DATA_BLOCK "PDI"   // DB129
{ S7_Optimized_Access := 'FALSE' }
VERSION : 0.0
// --------------------------------------------------------------------------------
// program:             PDI
// description :        automatically generated PDI
// name:                hp
// date        :        03.02.2021
// 
// revision:
// name:
// date:
//                     (c)CGS
// --------------------------------------------------------------------------------
   VAR
      CB_FLT_DC24V_K2 : Bool;   // HDI def M 72.0: fault circuit breakers DC 24V 1=OK
      CB_FLT_AC400V_K2 : Bool;   // HDI def M 72.1: fault circuit breakers AC 400V 1=OK
      SPARE_16_2 : Bool;   // HDI def M 72.4: spare digital input
      CB_FLT_AC230V : Bool;   // HDI def M 72.3: fault circuit breakers AC 230V 1=OK
      SPARE_16_4 : Bool;   // HDI def M 72.4: spare digital input
      SPARE_16_5 : Bool;   // HDI def M 72.5: spare digital input
      SPARE_16_6 : Bool;   // HDI def M 72.6: spare digital input
      SPARE_16_7 : Bool;   // HDI def M 72.7: spare digital input
      SPARE_17_0 : Bool;   // HDI def M 73.0: spare digital input
      UPS_24V_ALM : Bool;   // HDI def M 73.1: alarm dc-usv
      UPS_24V_NRM : Bool;   // HDI def M 73.2: main line ready buffered dc-usv
      EMO : Bool;   // HDI def M 73.3: Emergency off (1=ok)
      EMS : Bool;   // HDI def M 73.4: Emergency stop handling drives (1=ok)
      SPARE_17_5 : Bool;   // HDI def M 73.5: spare digital input
      SPARE_17_6 : Bool;   // HDI def M 73.6: spare digital input
      SPARE_17_7 : Bool;   // HDI def M 73.7: spare digital input
      P1_WRN : Bool;   // HDI def M 74.0: pump unit (P1) warning
      P1_FLT : Bool;   // HDI def M 74.1: pump unit (P1) error
      P1_IS_ON : Bool;   // HDI def M 74.2: pump unit (P1) running
      P1_WD : Bool;   // HDI def M 74.3: pump unit (P1) watchdog
      FIL_APS : Bool;   // HDI def M 74.4: pressure filter 1000 mbar
      MON_TMP_P2 : Bool;   // HDI def M 74.5: temperature monitoring P2
      MON_TMP_P1 : Bool;   // HDI def M 74.6: temperature monitoring P1
      SPARE_18_7 : Bool;   // HDI def M 74.7: spare digital input
      FCH_LFT_SDL_NUT : Bool;   // HDI def M 88.0: safety limit switch furnace chamber lift spindle nut
      LS_FCH_LFT_DN : Bool;   // HDI def M 88.1: limit switch furnace chamber lift down
      LS_FCH_HOOK_WORK : Bool;   // HDI def M 88.2: limit switch furnace chamber hook in working position
      LS_FCH_HOOK_HOME : Bool;   // HDI def M 88.3: limit switch furnace chamber hook in home position
      LS_TEC_FLG_DN : Bool;   // HDI def M 88.4: limit switch technolgy flange down
      TEC_FLG_SDL_NUT : Bool;   // HDI def M 88.5: safety limit switch technolgy flange lift spindle nut
      LS_V11_COV_OP : Bool;   // HDI def M 88.6: Cover V11 opened (isolation valve feeder)
      LS_V11_COV_CL : Bool;   // HDI def M 88.7: Cover V11 closed (isolation valve feeder)
      GCH_APS : Bool;   // HDI def M 89.0: pressure gate chamber 1000 mbar
      FCH_APS : Bool;   // HDI def M 89.1: pressure furnace chamber 1000 mbar
      FDR_APS : Bool;   // HDI def M 89.2: pressure feeder 1000 mbar
      FIL_2_APS : Bool;   // HDI def M 89.3: atmospheric pressure filter 2
      SPARE_33_4 : Bool;   // HDI def M 89.4: spare
      SPARE_33_5 : Bool;   // HDI def M 89.5: spare
      LS_V2_1_OP : Bool;   // HDI def M 89.6: valve position v2.1 fce chamber
      LS_V2_1_CL : Bool;   // HDI def M 89.7: valve position v2.1 fce chamber
      CB_FLT_AC400V_K5 : Bool;   // HDI def M 90.0: fault circuit breakers AC 400V +K5 1=OK
      CB_FLT_DC24V_K5 : Bool;   // HDI def M 90.1: fault circuit breakers DC 24V +K5 1=OK
      LS_MAG_LFT_UP : Bool;   // HDI def M 90.2: limit switch magnet lift up
      LS_MAG_LFT_DN : Bool;   // HDI def M 90.3: limit switch magnet lift down
      SLS_MAG_LFT : Bool;   // HDI def M 90.4: Safety limit switch magnet lift
      MAG_LFT_SDL_NUT1 : Bool;   // HDI def M 90.5: safety limit switch magnet lift spindle nut 1
      MAG_LFT_SDL_NUT2 : Bool;   // HDI def M 90.6: safety limit switch magnet lift spindle nut 2
      MAG_LFT_SDL_NUT3 : Bool;   // HDI def M 90.7: safety limit switch magnet lift spindle nut 3
      OIL_LVL_CR_SFT : Bool;   // HDI def M 91.0: Crucible shaft min. oil level
      LS_V1_OP : Bool;   // HDI def M 91.1: V1 opened
      LS_V1_CL : Bool;   // HDI def M 91.2: V1 closed
      MP_ENB_K5 : Bool;   // HDI def M 91.3: Mobile panel agree button +K5
      SLS_TEC_FLG_LFT : Bool;   // HDI def M 91.4: Safety limit switch technolgy flange lift
      SLS_FCH_LFT : Bool;   // HDI def M 91.5: Safety limit switch furnace chamber lift
      COMP_AIR_OK : Bool;   // HDI def M 91.6: pressure switch compressed air ok
      COMP_AIR_2_OK : Bool;   // HDI def M 91.7: pressure switch compressed air 2 (ACC) ok
      LS_V1_1_CL : Bool;   // HDI def M 105.0: limit switch valve v1.1 closed
      LS_V1_1_OP : Bool;   // HDI def M 105.1: limit switch valve v1.1 opened
      LS_V3_4_OP : Bool;   // HDI def M 105.2: limit switch valve v3.4 opened
      LS_V3_4_CL : Bool;   // HDI def M 105.3: limit switch valve v3.4 closed
      LS_V3_3_OP : Bool;   // HDI def M 105.4: limit switch valve v3.3 opened
      LS_V3_3_CL : Bool;   // HDI def M 105.5: limit switch valve v3.3 closed
      LS_V2_11_OP : Bool;   // HDI def M 105.6: limit switch valve v2.11 opened
      LS_V2_11_CL : Bool;   // HDI def M 105.7: limit switch valve v2.11 closed
      ACC_FCH_OV_PRS_1 : Bool;   // HDI def M 92.0: ACC furnace overpressure 1
      ACC_FCH_OV_PRS_2 : Bool;   // HDI def M 92.1: ACC furnace overpressure 2
      SPARE_48_2 : Bool;   // HDI def M 92.2: ACC spare
      ACC_WTR_FLW_OUT_OK : Bool;   // HDI def M 92.3: ACC output waterflow ok
      ACC_WTR_FLW_IN_OK : Bool;   // HDI def M 92.4: ACC input waterflow ok
      ACC_WTR_TMP_OUT_OK : Bool;   // HDI def M 92.5: ACC output watertemp. Ok
      OV_PRS_1_FLT : Bool;   // HDI def M 92.6: ACC overpressure 1 error/fault
      OV_PRS_2_FLT : Bool;   // HDI def M 92.7: ACC overpressure 2 error/fault
      ACC_SC_WTR_OK : Bool;   // HDI def M 93.0: ACC safety circuit
      ACC_SC_WTR_ATV : Bool;   // HDI def M 93.1: ACC safety circuit
      ACC_SC_HTR_OK : Bool;   // HDI def M 93.2: ACC safety circuit
      ACC_SC_HTR_ATV : Bool;   // HDI def M 93.3: ACC safety circuit
      ACC_KEY_RST : Bool;   // HDI def M 93.4: ACC reset key
      ACC_CB_FLT_DC24V : Bool;   // HDI def M 93.5: ACC 24V circuit breaker ok
      ACC_UPS_24V_ALM : Bool;   // HDI def M 93.6: ACC UPS OK Normal
      ACC_UPS_24V_NRM : Bool;   // HDI def M 93.7: ACC UPS Alarm
      DPH_RPT_DET_OK : Bool;   // HDI def M 94.0: ACC Diaphraghm rupture detector OK
      ACC_CB_FLT_AC230V : Bool;   // HDI def M 94.1: Fault circuit breakers AC 230V
      SPARE_90_2 : Bool;   // HDI def M 94.2: ACC spare
      SPARE_90_3 : Bool;   // HDI def M 94.3: ACC spare
      SPARE_90_4 : Bool;   // HDI def M 94.4: ACC spare
      SPARE_90_5 : Bool;   // HDI def M 94.5: ACC spare
      SPARE_90_6 : Bool;   // HDI def M 94.6: ACC spare
      SPARE_90_7 : Bool;   // HDI def M 94.7: ACC spare
      FU_P2_RDY : Bool;   // HDI def M 104.0: Frequency converter P2 ready/ no fault
      SPARE_144_1 : Bool;   // HDI def M 104.1: spare digital input
      SPARE_144_2 : Bool;   // HDI def M 104.2: spare digital input
      SPARE_144_3 : Bool;   // HDI def M 104.3: spare digital input
      SPARE_144_4 : Bool;   // HDI def M 104.4: spare digital input
      SPARE_144_5 : Bool;   // HDI def M 104.5: spare digital input
      SPARE_144_6 : Bool;   // HDI def M 104.6: spare digital input
      SPARE_144_7 : Bool;   // HDI def M 104.7: spare digital input
      LS_GCH_UP : Bool;   // HDI def M 95.0: limit switch gate chamber in upper position
      LS_GCH_DN : Bool;   // HDI def M 95.1: limit switch gate chamber in lower position
      LS_GCH_SW_IN : Bool;   // HDI def M 95.2: limit switch gate chamber swivelled in
      LS_GCH_SW_CLN : Bool;   // HDI def M 95.3: limit switch gate chamber swivelled in cleaning pos
      LS_GCH_SW_OUT : Bool;   // HDI def M 95.4: limit switch gate chamber swivelled out
      LS_GCH_SW_LOCK : Bool;   // HDI def M 95.5: limit switch gate chamber swivel locked
      SLS_GCH_LFT : Bool;   // HDI def M 95.6: Safety limit switch gate chamber lift
      LS_TCH_UP : Bool;   // HDI def M 95.7: limit switch top chamber in upper position
      LS_TCH_DN : Bool;   // HDI def M 96.0: limit switch top chamber in lower position
      LS_TCH_SW_IN : Bool;   // HDI def M 96.1: limit switch top chamber swivelled in
      LS_TCH_SW_CLN : Bool;   // HDI def M 96.2: limit switch top chamber swivelled in cleaning pos
      LS_TCH_SW_OUT : Bool;   // HDI def M 96.3: limit switch top chamber swivelled out
      LS_TCH_SW_LOCK : Bool;   // HDI def M 96.4: limit switch top chamber swivel locked
      LS_TCH_TILT_0 : Bool;   // HDI def M 96.5: limit switch top chamber tilt 0?horizental
      LS_TCH_TILT_30 : Bool;   // HDI def M 96.6: limit switch top chamber tilt 30?Cleaning position
      KEY_XT_LFT_SRV : Bool;   // HDI def M 96.7: Key switch service mode crystal lift
      LS_V7_UP : Bool;   // HDI def M 97.0: limit switch gate valve V7 in upper position
      LS_V7_DN : Bool;   // HDI def M 97.1: limit switch gate valve V7 in lower position
      LS_V7_SW_IN : Bool;   // HDI def M 97.2: limit switch gate valve V7 swiveled in
      LS_V7_SW_OUT : Bool;   // HDI def M 97.3: limit switch gate valve V7 swiveled out
      LS_V7_FLP_OP : Bool;   // HDI def M 97.4: limit switch gate valve V7 flap open
      LS_V7_CLN_POS : Bool;   // HDI def M 97.5: limit switch gate valve V7 in cleaning position
      LS_GCH_BEL_UP : Bool;   // HDI def M 97.6: limit switch gate chamber bellow in upper position
      LS_GCH_BEL_DN : Bool;   // HDI def M 97.7: limit switch gate chamber bellow in lower position
      LS_XT_SLID_BW : Bool;   // HDI def M 98.0: limit switch crystal handling slider in home position
      LS_XT_SLID_FW : Bool;   // HDI def M 98.1: limit switch crystal handling slider in work position
      LS_XT_SLID_MID : Bool;   // HDI def M 98.2: limit switch crystal handling slider in middle position
      LS_XT_CLP_CON : Bool;   // HDI def M 98.3: limit switch crystal handling clamps connected
      LS_XT_TILT_90 : Bool;   // HDI def M 98.4: limit switch crystal handling tilt in 90?
      LS_XT_TILT_75 : Bool;   // HDI def M 98.5: limit switch crystal handling tilt in 75?
      LS_UP_XT_CLP_FLT : Bool;   // HDI def M 98.6: limit switch upper crystal clamp fault
      SPARE_275_7 : Bool;   // HDI def M 98.7: spare digital input
      LS_UP_XT_CLP_OP : Bool;   // HDI def M 99.0: limit switch upper crystal clamp open
      LS_UP_XT_CLP_CL : Bool;   // HDI def M 99.1: limit switch upper crystal clamp closed
      LS_UP_XT_CLP_SAVE : Bool;   // HDI def M 99.2: limit switch upper crystal clamp save
      LS_UP_XT_CLP_PLATE : Bool;   // HDI def M 99.3: limit switch upper crystal clamp plate
      LS_LO_XT_CLP_FLT : Bool;   // HDI def M 99.4: limit switch lower crystal clamp fault
      LS_LO_XT_CLP_OP : Bool;   // HDI def M 99.5: limit switch lower crystal clamp open
      LS_LO_XT_CLP_CL : Bool;   // HDI def M 99.6: limit switch lower crystal clamp closed
      LS_LO_XT_CLP_SAVE : Bool;   // HDI def M 99.7: limit switch lower crystal clamp save
      LS_LO_XT_CLP_PLATE : Bool;   // HDI def M 100.0: limit switch upper crystal clamp plate
      LS_HOI_TOOL_INST : Bool;   // HDI def M 100.1: limit switch HOI tool installed
      XT_DRP_OUT_PRT_1_CL : Bool;   // HDI def M 100.2: crystal drop out protection 1 closed (upper left side)
      XT_DRP_OUT_PRT_1_OP : Bool;   // HDI def M 100.3: crystal drop out protection 1 opened (upper left side)
      XT_DRP_OUT_PRT_2_CL : Bool;   // HDI def M 100.4: crystal drop out protection 2 closed (upper right side)
      XT_DRP_OUT_PRT_2_OP : Bool;   // HDI def M 100.5: crystal drop out protection 2 opened (upper right side)
      CB_FLT_AC400V_K8 : Bool;   // HDI def M 100.6: fault circuit breakers AC 400V 1=OK
      CB_FLT_DC24V_K8 : Bool;   // HDI def M 100.7: fault circuit breakers DC 24V 1=OK
      XT_DRP_OUT_PRT_3_CL : Bool;   // HDI def M 101.0: crystal drop out protection 3 closed (lower left side)
      XT_DRP_OUT_PRT_3_OP : Bool;   // HDI def M 101.1: crystal drop out protection 3 opened (lower left side)
      XT_DRP_OUT_PRT_4_CL : Bool;   // HDI def M 101.2: crystal drop out protection 4 closed (lower right side)
      XT_DRP_OUT_PRT_4_OP : Bool;   // HDI def M 101.3: crystal drop out protection 4 opened (lower right side)
      LS_XT_HDL_SW_UNLOCK : Bool;   // HDI def M 101.4: limit switch crystal handling swivel unlocked
      LS_XT_HDL_SW_LOCK : Bool;   // HDI def M 101.5: limit switch crystal handling swivel locked 145?
      LS_GCH_DOOR_OP : Bool;   // HDI def M 101.6: limit switch gate chamber door opened
      LS_GCH_DOOR_CL : Bool;   // HDI def M 101.7: limit switch gate chamber door closed
      MCC_CONTACT_XT : Bool;   // HDI def M 102.0: seed contact detection (xt isolated)
      OIL_LVL_XT_SFT : Bool;   // HDI def M 102.1: Crystal shaft min. oil level
      LS_XT_SFT_SRV_POS : Bool;   // HDI def M 102.2: limit switch crystal shaft service position
      LS_XT_TOP_POS : Bool;   // HDI def M 102.3: limit switch crystal shaft in top position
      SLS_TCH_LFT : Bool;   // HDI def M 102.4: Safety limit switch top chamber lift
      XT_ROT_CAM_TRG : Bool;   // HDI def M 102.5: limit switch xtal rotation camera trigger
      MP_ENB_K8 : Bool;   // HDI def M 102.6: Mobile panel agree button +K8
      MP_ENB_K9 : Bool;   // HDI def M 102.7: Mobile panel agree button +K9
      LS_V3_OP : Bool;   // HDI def M 103.0: valve position V3 open
      LS_V3_CL : Bool;   // HDI def M 103.1: Valve position V3 closed
      FDR_LS_V3_2_OP : Bool;   // HDI def M 103.2: valve position V3_2 open
      FDR_LS_V3_2_CL : Bool;   // HDI def M 103.3: Valve position V3_2 closed
      LSR_SEN_OBJ_DET : Bool;   // HDI def M 103.4: spare digital input
      SPARE_280_5 : Bool;   // HDI def M 103.5: spare digital input
      SPARE_280_6 : Bool;   // HDI def M 103.6: spare digital input
      SPARE_280_7 : Bool;   // HDI def M 103.7: spare digital input
      LS_V11_OP : Bool;   // HDI def M 89.3: V 11 open (isolation valve feeder)
      LS_V11_CL : Bool;   // HDI def M 89.4: V 11 closed (isolation valve feeder)
      FDR_HOP_CON : Bool;   // HDI def M 89.5: hopper connected to feeder
   END_VAR
BEGIN
END_DATA_BLOCK

DATA_BLOCK "PDO"   // DB130
{ S7_Optimized_Access := 'FALSE' }
VERSION : 0.0
// --------------------------------------------------------------------------------
// program:             PDO
// description :        automatically generated PDO
// name:                hp
// date        :        03.02.2021
// 
// revision:
// name:
// date:
//                     (c)CGS
// --------------------------------------------------------------------------------
   VAR
      HOR_OPP_K2 : Bool;   // HDO def M 136.0: Horn +K2
      LMP_RD_K2 : Bool;   // HDO def M 136.1: Lamp red +K2
      LMP_YE_K2 : Bool;   // HDO def M 136.2: Lamp yellow +K2
      LMP_GN_K2 : Bool;   // HDO def M 136.3: Lamp green +K2
      LMP_BU_K2 : Bool;   // HDO def M 136.4: Lamp blue +K2
      HOR_MAG_ACTIVE : Bool;   // HDO def M 136.5: Horn magnet active( Lift)
      LMP_MAG_ACTIVE : Bool;   // HDO def M 136.6: Lamp magnet active( Lift+ Field on)
      SPARE_16_7 : Bool;   // HDO def M 136.7: spare digital output
      P1_ON : Bool;   // HDO def M 137.0: Vacuum pump 1 on (furnace chamber)
      P3_ON : Bool;   // HDO def M 137.1: Vacuum pump 3 on (gate chamber)
      P2_ON : Bool;   // HDO def M 137.2: Vacuum pump 2 on (roots furnace chamber)
      P1_SEAL_GAS : Bool;   // HDO def M 137.3: Vacuum pump 1 seal gas on
      P3_SEAL_GAS : Bool;   // HDO def M 137.4: Vacuum pump 3 seal gas on
      HTR_PWR_ON : Bool;   // HDO def M 137.4: Heater power supply on
      V10 : Bool;   // HDO def M 137.6: Vacuum pump 1 secuvac valve V10 on
      MON_TMP_P2_RES : Bool;   // HDO def M 137.7: temperature monitoring pump 2 reset
      SPARE_18_0 : Bool;   // HDO def M 138.0: spare digital output
      SPARE_18_1 : Bool;   // HDO def M 138.1: spare digital output
      SPARE_18_2 : Bool;   // HDO def M 138.2: spare digital output
      SPARE_18_3 : Bool;   // HDO def M 138.3: spare digital output
      SPARE_18_4 : Bool;   // HDO def M 138.4: spare digital output
      SPARE_18_5 : Bool;   // HDO def M 138.5: spare digital output
      SPARE_18_6 : Bool;   // HDO def M 138.6: spare digital output
      SPARE_18_7 : Bool;   // HDO def M 138.7: spare digital output
      V1_OP : Bool;   // HDO def M 142.0: V1 open
      V1_CL : Bool;   // HDO def M 142.1: V1 close
      SPARE_32_2 : Bool;   // HDO def M 142.2: spare digital output
      SPARE_32_3 : Bool;   // HDO def M 142.3: spare digital output
      SPARE_32_4 : Bool;   // HDO def M 142.4: spare digital output
      CR_ROT_ENB : Bool;   // HDO def M 142.5: controller enable crucible rotation
      CR_LFT_ENB : Bool;   // HDO def M 142.6: controller enable crucible lift
      FU_FCB_HDL_ON : Bool;   // HDO def M 142.7: Frequency converter FCB handling on
      TEC_FLG_LFT_ENB : Bool;   // HDO def M 143.0: controller enable techn chamber lift
      FCH_LFT_ENB : Bool;   // HDO def M 143.1: controller enable lower chamber parts lift
      MAG_LFT_UP : Bool;   // HDO def M 143.2: Magnet lift drive upwards
      MAG_LFT_DN : Bool;   // HDO def M 143.3: Magnet lift drive downwards
      BRK_MAG_LFT : Bool;   // HDO def M 143.4: Brake magnet lift
      SPARE_33_5 : Bool;   // HDO def M 143.5: spare digital output
      SPARE_33_6 : Bool;   // HDO def M 143.6: spare digital output
      SPARE_33_7 : Bool;   // HDO def M 143.7: spare digital output
      V1_1_OP : Bool;   // HDO def M 144.0: V1.1 open
      V1_1_CL : Bool;   // HDO def M 144.1: V1.1 close
      SPARE_34_2 : Bool;   // HDO def M 144.2: spare digital output
      SPARE_34_3 : Bool;   // HDO def M 144.3: spare digital output
      SPARE_34_4 : Bool;   // HDO def M 144.4: spare digital output
      SPARE_34_5 : Bool;   // HDO def M 144.5: spare digital output
      SPARE_34_6 : Bool;   // HDO def M 144.6: spare digital output
      SPARE_34_7 : Bool;   // HDO def M 144.7: spare digital output
      ACC_SC_HTR_STR : Bool;   // HDO def M 146.0: ACC Heizung START
      ACC_SC_HTR_RST : Bool;   // HDO def M 146.1: ACC Heizung RESET
      ACC_SC_WTR_STR : Bool;   // HDO def M 146.2: ACC K黨lwasser START
      ACC_SC_WTR_RST : Bool;   // HDO def M 146.3: ACC K黨lwasser RESET
      ACC_ALM_LT_1 : Bool;   // HDO def M 146.4: ACC Blitzlicht Kasten
      ACC_ALM_SND_1 : Bool;   // HDO def M 146.5: ACC Sirene Kasten
      ACC_ALM_LT_2 : Bool;   // HDO def M 146.6: ACC Blitzlicht Bedienpult
      ACC_ALM_SND_2 : Bool;   // HDO def M 146.7: ACC Sirene Bedienpult
      FCH_HOOK_HOME : Bool;   // HDO def M 150.0: Valve block lower furnace chamber hook unlocking
      FCH_HOOK_WORK : Bool;   // HDO def M 150.1: Valve block lower furnace chamber hook locking
      UP_FCH_SW_BRK : Bool;   // HDO def M 150.2: Valve block upper chamber swivel release brake
      LO_FCH_SW_BRK : Bool;   // HDO def M 150.3: Valve block lower chamber swivel release brake
      TEC_FLG_SW_BRK : Bool;   // HDO def M 150.4: Valve block tech. flange swivel release brake
      V25 : Bool;   // HDO def M 150.5: Valve block argon inlet pressure storage tank, V25 open
      V2_1 : Bool;   // HDO def M 150.6: Valve block vacuum valve, V2.1 open
      V21 : Bool;   // HDO def M 150.7: Valve block air valve vacuum pipe, V21+V21.1 open
      V19 : Bool;   // HDO def M 151.0: Valve block extraktion valve filter, V19 open
      V20 : Bool;   // HDO def M 151.1: Valve block air valve filter, V20 open
      V22 : Bool;   // HDO def M 151.2: Valve block argon valve filter, V22 open
      V9_2 : Bool;   // HDO def M 151.3: Valve block ventiliation valve vaccum line gate, V9_2
      V22_1 : Bool;   // HDO def M 151.4: Valve block argon valve bypass filter, V22.1 open
      V3_4 : Bool;   // HDO def M 151.5: Valve block vacuum valve, V3.4 open
      V3_3 : Bool;   // HDO def M 151.6: Valve block vacuum valve, V3.3 open
      V2_11 : Bool;   // HDO def M 151.7: Valve block vacuum valve, V2.11 open
      P2_FU_ON : Bool;   // HDO def M 152.0: Frequency converter P2 start
      P2_FU_RES : Bool;   // HDO def M 152.1: Frequency converter P2 fault reset
      SPARE_144_2 : Bool;   // HDO def M 152.2: spare digital output
      SPARE_144_3 : Bool;   // HDO def M 152.3: spare digital output
      SPARE_144_4 : Bool;   // HDO def M 152.4: spare digital output
      SPARE_144_5 : Bool;   // HDO def M 152.5: spare digital output
      SPARE_144_6 : Bool;   // HDO def M 152.6: spare digital output
      SPARE_144_7 : Bool;   // HDO def M 152.7: spare digital output
      V4 : Bool;   // HDO def M 150.0: Valve block V4 valve argon gas inlet (gate chamber)
      V5 : Bool;   // HDO def M 150.1: Valve block V5 valve argon gas inlet controlled (gch)
      V6 : Bool;   // HDO def M 150.2: Valve block V6 valve argon gas inlet controlled (Fch)
      V3 : Bool;   // HDO def M 150.3: Valve block V3 vacuum valve (gate chamber)
      V3_2 : Bool;   // HDO def M 150.4: Valve block V3.2 vacuum valve feeder
      V24 : Bool;   // HDO def M 150.5: Valve block V24 valve argon gas inlet feeder
      XT_DRP_OUT_PRT_CL : Bool;   // HDO def M 150.6: Valve block close crystal drop out protection
      XT_DRP_OUT_PRT_OP : Bool;   // HDO def M 150.7: Valve block open crystal drop out protection
      TCH_SW_LOCK : Bool;   // HDO def M 151.0: Valve block top chamber swivel lock close
      TCH_SW_UNLOCK : Bool;   // HDO def M 151.1: Valve block top chamber swivel lock open
      GCH_SW_LOCK : Bool;   // HDO def M 151.2: Valve block gate chamber swivel lock close
      GCH_SW_UNLOCK : Bool;   // HDO def M 151.3: Valve block gate chamber swivel lock open
      XT_HDL_SW_LOCK : Bool;   // HDO def M 151.4: Valve block xtal handling swivel lock close (145?
      XT_HDL_SW_UNLOCK : Bool;   // HDO def M 151.5: Valve block xtal handling swivel lock open (145?
      FDR_V11_OP : Bool;   // HDO def M 151.6: Valve block open V11 (isolation valve feeder)
      FDR_V11_CL : Bool;   // HDO def M 151.7: Valve block close V11 (isolation valve feeder)
      FDR_V11_CVR_OP : Bool;   // HDO def M 152.0: Valve block open cover V11 (isolation valve feeder)
      FDR_V11_CVR_CL : Bool;   // HDO def M 152.1: Valve block close cover V11 (isolation valve feeder)
      SPARE_226_2 : Bool;   // HDO def M 152.2: Valve block spare output
      SPARE_226_3 : Bool;   // HDO def M 152.3: Valve block spare output
      SPARE_226_4 : Bool;   // HDO def M 152.4: Valve block spare output
      SPARE_226_5 : Bool;   // HDO def M 152.5: Valve block spare output
      SPARE_226_6 : Bool;   // HDO def M 152.6: Valve block spare output
      SPARE_226_7 : Bool;   // HDO def M 152.7: Valve block spare output
      HOR_OPP_K8 : Bool;   // HDO def M 160.0: Horn +K8
      LMP_RD_K8 : Bool;   // HDO def M 160.1: Lamp red +K8
      LMP_YE_K8 : Bool;   // HDO def M 160.2: Lamp yellow +K8
      LMP_GN_K8 : Bool;   // HDO def M 160.3: Lamp green +K8
      LMP_BU_K8 : Bool;   // HDO def M 160.4: Lamp blue +K8
      XT_ROT_ENB : Bool;   // HDO def M 160.5: controller enable crystal rotation
      XT_LFT_ENB : Bool;   // HDO def M 160.6: controller enable crystal lift
      XT_HDL_LFT_ENB : Bool;   // HDO def M 160.7: controller enable crystal handling lift
      XT_HDL_SW_ENB : Bool;   // HDO def M 161.0: controller enable crystal handling swivel
      FU_GCB_HDL_ON : Bool;   // HDO def M 161.1: Frequency converter GCB handling on
      LSR_SEN_PWR_ON : Bool;   // HDO def M 161.2: supply voltage for laser sensor on
      SPARE_273_3 : Bool;   // HDO def M 161.3: spare digital output
      SPARE_273_4 : Bool;   // HDO def M 161.4: spare digital output
      SPARE_273_5 : Bool;   // HDO def M 161.5: spare digital output
      XT_HDL_SLID_FW : Bool;   // HDO def M 161.6: Motor crystal handling slider forwards
      XT_HDL_SLID_BW : Bool;   // HDO def M 161.7: Motor crystal handling slider backwards
      XT_CLP_TILT_BW : Bool;   // HDO def M 163.0: Motor crystal clamp tilt backwards
      XT_CLP_TILT_FW : Bool;   // HDO def M 163.1: Motor crystal clamp tilt forwards (75?
      XT_CLP_TILT_BRK : Bool;   // HDO def M 163.2: Motor crystal clamp tilt brake
      XT_CLP_ABV_OP : Bool;   // HDO def M 163.3: Motor crystal clamp above open
      XT_CLP_ABV_CL : Bool;   // HDO def M 163.4: Motor crystal clamp above close
      XT_CLP_ABV_BRK : Bool;   // HDO def M 163.5: Brake crystal clamp above
      XT_CLP_ABV_RST : Bool;   // HDO def M 163.6: Reset controller crystal clamp above
      GCH_LFT_ENB : Bool;   // HDO def M 163.7: controller enable gate chamber lift
      XT_CLP_BLW_OP : Bool;   // HDO def M 164.0: Motor crystal clamp below open
      XT_CLP_BLW_CL : Bool;   // HDO def M 164.1: Motor crystal clamp below close
      XT_CLP_BLW_BRK : Bool;   // HDO def M 164.2: Brake crystal clamp below
      XT_CLP_BLW_RST : Bool;   // HDO def M 164.3: Reset controller crystal clamp below
      MCC_TEST_XT : Bool;   // HDO def M 164.4: seed contact detection test output ( xt isolated)
      MCC_ENB_XT : Bool;   // HDO def M 164.5: seed contact detection enable output (xt isolated)
      TCH_LFT_ENB : Bool;   // HDO def M 164.6: controller enable top chamber lift
      TCH_TILT_ENB : Bool;   // HDO def M 164.7: controller enable top chamber tilt
      GTE_V_LFT_ENB : Bool;   // HDO def M 165.0: controller enable gate valve lift
      GTE_V_SW_ENB : Bool;   // HDO def M 165.1: controller enable gate valve swivel
      BEL_LFT_ENB : Bool;   // HDO def M 165.2: controller enable gate bellow lift
      HOR_OPP_K9 : Bool;   // HDO def M 165.3: Horn +K9
      LMP_RD_K9 : Bool;   // HDO def M 165.4: Lamp red +K9
      LMP_YE_K9 : Bool;   // HDO def M 165.5: Lamp yellow +K9
      LMP_GN_K9 : Bool;   // HDO def M 165.6: Lamp green +K9
      LMP_BU_K9 : Bool;   // HDO def M 165.7: Lamp blue +K9
   END_VAR
BEGIN
END_DATA_BLOCK

DATA_BLOCK "SDI"   // DB131
{ S7_Optimized_Access := 'FALSE' }
VERSION : 0.0
// --------------------------------------------------------------------------------
// program:             SDI
// description :        automatically generated SDI
// name:                hp
// date        :        03.02.2021
// 
// revision:
// name:
// date:
//                     (c)CGS
// --------------------------------------------------------------------------------
   VAR
      CB_FLT_DC24V_K2 : Bool;   // HDI def M 72.0: fault circuit breakers DC 24V 1=OK
      CB_FLT_AC400V_K2 : Bool;   // HDI def M 72.1: fault circuit breakers AC 400V 1=OK
      SPARE_16_2 : Bool;   // HDI def M 72.4: spare digital input
      CB_FLT_AC230V : Bool;   // HDI def M 72.3: fault circuit breakers AC 230V 1=OK
      SPARE_16_4 : Bool;   // HDI def M 72.4: spare digital input
      SPARE_16_5 : Bool;   // HDI def M 72.5: spare digital input
      SPARE_16_6 : Bool;   // HDI def M 72.6: spare digital input
      SPARE_16_7 : Bool;   // HDI def M 72.7: spare digital input
      SPARE_17_0 : Bool;   // HDI def M 73.0: spare digital input
      UPS_24V_ALM : Bool;   // HDI def M 73.1: alarm dc-usv
      UPS_24V_NRM : Bool;   // HDI def M 73.2: main line ready buffered dc-usv
      EMO : Bool;   // HDI def M 73.3: Emergency off (1=ok)
      EMS : Bool;   // HDI def M 73.4: Emergency stop handling drives (1=ok)
      SPARE_17_5 : Bool;   // HDI def M 73.5: spare digital input
      SPARE_17_6 : Bool;   // HDI def M 73.6: spare digital input
      SPARE_17_7 : Bool;   // HDI def M 73.7: spare digital input
      P1_WRN : Bool;   // HDI def M 74.0: pump unit (P1) warning
      P1_FLT : Bool;   // HDI def M 74.1: pump unit (P1) error
      P1_IS_ON : Bool;   // HDI def M 74.2: pump unit (P1) running
      P1_WD : Bool;   // HDI def M 74.3: pump unit (P1) watchdog
      FIL_APS : Bool;   // HDI def M 74.4: pressure filter 1000 mbar
      MON_TMP_P2 : Bool;   // HDI def M 74.5: temperature monitoring P2
      MON_TMP_P1 : Bool;   // HDI def M 74.6: temperature monitoring P1
      SPARE_18_7 : Bool;   // HDI def M 74.7: spare digital input
      FCH_LFT_SDL_NUT : Bool;   // HDI def M 88.0: safety limit switch furnace chamber lift spindle nut
      LS_FCH_LFT_DN : Bool;   // HDI def M 88.1: limit switch furnace chamber lift down
      LS_FCH_HOOK_WORK : Bool;   // HDI def M 88.2: limit switch furnace chamber hook in working position
      LS_FCH_HOOK_HOME : Bool;   // HDI def M 88.3: limit switch furnace chamber hook in home position
      LS_TEC_FLG_DN : Bool;   // HDI def M 88.4: limit switch technolgy flange down
      TEC_FLG_SDL_NUT : Bool;   // HDI def M 88.5: safety limit switch technolgy flange lift spindle nut
      LS_V11_COV_OP : Bool;   // HDI def M 88.6: Cover V11 opened (isolation valve feeder)
      LS_V11_COV_CL : Bool;   // HDI def M 88.7: Cover V11 closed (isolation valve feeder)
      GCH_APS : Bool;   // HDI def M 89.0: pressure gate chamber 1000 mbar
      FCH_APS : Bool;   // HDI def M 89.1: pressure furnace chamber 1000 mbar
      FDR_APS : Bool;   // HDI def M 89.2: pressure feeder 1000 mbar
      FIL_2_APS : Bool;   // HDI def M 89.3: atmospheric pressure filter 2
      SPARE_33_4 : Bool;   // HDI def M 89.4: spare
      SPARE_33_5 : Bool;   // HDI def M 89.5: spare
      LS_V2_1_OP : Bool;   // HDI def M 89.6: valve position v2.1 fce chamber
      LS_V2_1_CL : Bool;   // HDI def M 89.7: valve position v2.1 fce chamber
      CB_FLT_AC400V_K5 : Bool;   // HDI def M 90.0: fault circuit breakers AC 400V +K5 1=OK
      CB_FLT_DC24V_K5 : Bool;   // HDI def M 90.1: fault circuit breakers DC 24V +K5 1=OK
      LS_MAG_LFT_UP : Bool;   // HDI def M 90.2: limit switch magnet lift up
      LS_MAG_LFT_DN : Bool;   // HDI def M 90.3: limit switch magnet lift down
      SLS_MAG_LFT : Bool;   // HDI def M 90.4: Safety limit switch magnet lift
      MAG_LFT_SDL_NUT1 : Bool;   // HDI def M 90.5: safety limit switch magnet lift spindle nut 1
      MAG_LFT_SDL_NUT2 : Bool;   // HDI def M 90.6: safety limit switch magnet lift spindle nut 2
      MAG_LFT_SDL_NUT3 : Bool;   // HDI def M 90.7: safety limit switch magnet lift spindle nut 3
      OIL_LVL_CR_SFT : Bool;   // HDI def M 91.0: Crucible shaft min. oil level
      LS_V1_OP : Bool;   // HDI def M 91.1: V1 opened
      LS_V1_CL : Bool;   // HDI def M 91.2: V1 closed
      MP_ENB_K5 : Bool;   // HDI def M 91.3: Mobile panel agree button +K5
      SLS_TEC_FLG_LFT : Bool;   // HDI def M 91.4: Safety limit switch technolgy flange lift
      SLS_FCH_LFT : Bool;   // HDI def M 91.5: Safety limit switch furnace chamber lift
      COMP_AIR_OK : Bool;   // HDI def M 91.6: pressure switch compressed air ok
      COMP_AIR_2_OK : Bool;   // HDI def M 91.7: pressure switch compressed air 2 (ACC) ok
      LS_V1_1_CL : Bool;   // HDI def M 105.0: limit switch valve v1.1 closed
      LS_V1_1_OP : Bool;   // HDI def M 105.1: limit switch valve v1.1 opened
      LS_V3_4_OP : Bool;   // HDI def M 105.2: limit switch valve v3.4 opened
      LS_V3_4_CL : Bool;   // HDI def M 105.3: limit switch valve v3.4 closed
      LS_V3_3_OP : Bool;   // HDI def M 105.4: limit switch valve v3.3 opened
      LS_V3_3_CL : Bool;   // HDI def M 105.5: limit switch valve v3.3 closed
      LS_V2_11_OP : Bool;   // HDI def M 105.6: limit switch valve v2.11 opened
      LS_V2_11_CL : Bool;   // HDI def M 105.7: limit switch valve v2.11 closed
      ACC_FCH_OV_PRS_1 : Bool;   // HDI def M 92.0: ACC furnace overpressure 1
      ACC_FCH_OV_PRS_2 : Bool;   // HDI def M 92.1: ACC furnace overpressure 2
      SPARE_48_2 : Bool;   // HDI def M 92.2: ACC spare
      ACC_WTR_FLW_OUT_OK : Bool;   // HDI def M 92.3: ACC output waterflow ok
      ACC_WTR_FLW_IN_OK : Bool;   // HDI def M 92.4: ACC input waterflow ok
      ACC_WTR_TMP_OUT_OK : Bool;   // HDI def M 92.5: ACC output watertemp. Ok
      OV_PRS_1_FLT : Bool;   // HDI def M 92.6: ACC overpressure 1 error/fault
      OV_PRS_2_FLT : Bool;   // HDI def M 92.7: ACC overpressure 2 error/fault
      ACC_SC_WTR_OK : Bool;   // HDI def M 93.0: ACC safety circuit
      ACC_SC_WTR_ATV : Bool;   // HDI def M 93.1: ACC safety circuit
      ACC_SC_HTR_OK : Bool;   // HDI def M 93.2: ACC safety circuit
      ACC_SC_HTR_ATV : Bool;   // HDI def M 93.3: ACC safety circuit
      ACC_KEY_RST : Bool;   // HDI def M 93.4: ACC reset key
      ACC_CB_FLT_DC24V : Bool;   // HDI def M 93.5: ACC 24V circuit breaker ok
      ACC_UPS_24V_ALM : Bool;   // HDI def M 93.6: ACC UPS OK Normal
      ACC_UPS_24V_NRM : Bool;   // HDI def M 93.7: ACC UPS Alarm
      DPH_RPT_DET_OK : Bool;   // HDI def M 94.0: ACC Diaphraghm rupture detector OK
      ACC_CB_FLT_AC230V : Bool;   // HDI def M 94.1: Fault circuit breakers AC 230V
      SPARE_90_2 : Bool;   // HDI def M 94.2: ACC spare
      SPARE_90_3 : Bool;   // HDI def M 94.3: ACC spare
      SPARE_90_4 : Bool;   // HDI def M 94.4: ACC spare
      SPARE_90_5 : Bool;   // HDI def M 94.5: ACC spare
      SPARE_90_6 : Bool;   // HDI def M 94.6: ACC spare
      SPARE_90_7 : Bool;   // HDI def M 94.7: ACC spare
      FU_P2_RDY : Bool;   // HDI def M 104.0: Frequency converter P2 ready/ no fault
      SPARE_144_1 : Bool;   // HDI def M 104.1: spare digital input
      SPARE_144_2 : Bool;   // HDI def M 104.2: spare digital input
      SPARE_144_3 : Bool;   // HDI def M 104.3: spare digital input
      SPARE_144_4 : Bool;   // HDI def M 104.4: spare digital input
      SPARE_144_5 : Bool;   // HDI def M 104.5: spare digital input
      SPARE_144_6 : Bool;   // HDI def M 104.6: spare digital input
      SPARE_144_7 : Bool;   // HDI def M 104.7: spare digital input
      LS_GCH_UP : Bool;   // HDI def M 95.0: limit switch gate chamber in upper position
      LS_GCH_DN : Bool;   // HDI def M 95.1: limit switch gate chamber in lower position
      LS_GCH_SW_IN : Bool;   // HDI def M 95.2: limit switch gate chamber swivelled in
      LS_GCH_SW_CLN : Bool;   // HDI def M 95.3: limit switch gate chamber swivelled in cleaning pos
      LS_GCH_SW_OUT : Bool;   // HDI def M 95.4: limit switch gate chamber swivelled out
      LS_GCH_SW_LOCK : Bool;   // HDI def M 95.5: limit switch gate chamber swivel locked
      SLS_GCH_LFT : Bool;   // HDI def M 95.6: Safety limit switch gate chamber lift
      LS_TCH_UP : Bool;   // HDI def M 95.7: limit switch top chamber in upper position
      LS_TCH_DN : Bool;   // HDI def M 96.0: limit switch top chamber in lower position
      LS_TCH_SW_IN : Bool;   // HDI def M 96.1: limit switch top chamber swivelled in
      LS_TCH_SW_CLN : Bool;   // HDI def M 96.2: limit switch top chamber swivelled in cleaning pos
      LS_TCH_SW_OUT : Bool;   // HDI def M 96.3: limit switch top chamber swivelled out
      LS_TCH_SW_LOCK : Bool;   // HDI def M 96.4: limit switch top chamber swivel locked
      LS_TCH_TILT_0 : Bool;   // HDI def M 96.5: limit switch top chamber tilt 0?horizental
      LS_TCH_TILT_30 : Bool;   // HDI def M 96.6: limit switch top chamber tilt 30?Cleaning position
      KEY_XT_LFT_SRV : Bool;   // HDI def M 96.7: Key switch service mode crystal lift
      LS_V7_UP : Bool;   // HDI def M 97.0: limit switch gate valve V7 in upper position
      LS_V7_DN : Bool;   // HDI def M 97.1: limit switch gate valve V7 in lower position
      LS_V7_SW_IN : Bool;   // HDI def M 97.2: limit switch gate valve V7 swiveled in
      LS_V7_SW_OUT : Bool;   // HDI def M 97.3: limit switch gate valve V7 swiveled out
      LS_V7_FLP_OP : Bool;   // HDI def M 97.4: limit switch gate valve V7 flap open
      LS_V7_CLN_POS : Bool;   // HDI def M 97.5: limit switch gate valve V7 in cleaning position
      LS_GCH_BEL_UP : Bool;   // HDI def M 97.6: limit switch gate chamber bellow in upper position
      LS_GCH_BEL_DN : Bool;   // HDI def M 97.7: limit switch gate chamber bellow in lower position
      LS_XT_SLID_BW : Bool;   // HDI def M 98.0: limit switch crystal handling slider in home position
      LS_XT_SLID_FW : Bool;   // HDI def M 98.1: limit switch crystal handling slider in work position
      LS_XT_SLID_MID : Bool;   // HDI def M 98.2: limit switch crystal handling slider in middle position
      LS_XT_CLP_CON : Bool;   // HDI def M 98.3: limit switch crystal handling clamps connected
      LS_XT_TILT_90 : Bool;   // HDI def M 98.4: limit switch crystal handling tilt in 90?
      LS_XT_TILT_75 : Bool;   // HDI def M 98.5: limit switch crystal handling tilt in 75?
      LS_UP_XT_CLP_FLT : Bool;   // HDI def M 98.6: limit switch upper crystal clamp fault
      SPARE_275_7 : Bool;   // HDI def M 98.7: spare digital input
      LS_UP_XT_CLP_OP : Bool;   // HDI def M 99.0: limit switch upper crystal clamp open
      LS_UP_XT_CLP_CL : Bool;   // HDI def M 99.1: limit switch upper crystal clamp closed
      LS_UP_XT_CLP_SAVE : Bool;   // HDI def M 99.2: limit switch upper crystal clamp save
      LS_UP_XT_CLP_PLATE : Bool;   // HDI def M 99.3: limit switch upper crystal clamp plate
      LS_LO_XT_CLP_FLT : Bool;   // HDI def M 99.4: limit switch lower crystal clamp fault
      LS_LO_XT_CLP_OP : Bool;   // HDI def M 99.5: limit switch lower crystal clamp open
      LS_LO_XT_CLP_CL : Bool;   // HDI def M 99.6: limit switch lower crystal clamp closed
      LS_LO_XT_CLP_SAVE : Bool;   // HDI def M 99.7: limit switch lower crystal clamp save
      LS_LO_XT_CLP_PLATE : Bool;   // HDI def M 100.0: limit switch upper crystal clamp plate
      LS_HOI_TOOL_INST : Bool;   // HDI def M 100.1: limit switch HOI tool installed
      XT_DRP_OUT_PRT_1_CL : Bool;   // HDI def M 100.2: crystal drop out protection 1 closed (upper left side)
      XT_DRP_OUT_PRT_1_OP : Bool;   // HDI def M 100.3: crystal drop out protection 1 opened (upper left side)
      XT_DRP_OUT_PRT_2_CL : Bool;   // HDI def M 100.4: crystal drop out protection 2 closed (upper right side)
      XT_DRP_OUT_PRT_2_OP : Bool;   // HDI def M 100.5: crystal drop out protection 2 opened (upper right side)
      CB_FLT_AC400V_K8 : Bool;   // HDI def M 100.6: fault circuit breakers AC 400V 1=OK
      CB_FLT_DC24V_K8 : Bool;   // HDI def M 100.7: fault circuit breakers DC 24V 1=OK
      XT_DRP_OUT_PRT_3_CL : Bool;   // HDI def M 101.0: crystal drop out protection 3 closed (lower left side)
      XT_DRP_OUT_PRT_3_OP : Bool;   // HDI def M 101.1: crystal drop out protection 3 opened (lower left side)
      XT_DRP_OUT_PRT_4_CL : Bool;   // HDI def M 101.2: crystal drop out protection 4 closed (lower right side)
      XT_DRP_OUT_PRT_4_OP : Bool;   // HDI def M 101.3: crystal drop out protection 4 opened (lower right side)
      LS_XT_HDL_SW_UNLOCK : Bool;   // HDI def M 101.4: limit switch crystal handling swivel unlocked
      LS_XT_HDL_SW_LOCK : Bool;   // HDI def M 101.5: limit switch crystal handling swivel locked 145?
      LS_GCH_DOOR_OP : Bool;   // HDI def M 101.6: limit switch gate chamber door opened
      LS_GCH_DOOR_CL : Bool;   // HDI def M 101.7: limit switch gate chamber door closed
      MCC_CONTACT_XT : Bool;   // HDI def M 102.0: seed contact detection (xt isolated)
      OIL_LVL_XT_SFT : Bool;   // HDI def M 102.1: Crystal shaft min. oil level
      LS_XT_SFT_SRV_POS : Bool;   // HDI def M 102.2: limit switch crystal shaft service position
      LS_XT_TOP_POS : Bool;   // HDI def M 102.3: limit switch crystal shaft in top position
      SLS_TCH_LFT : Bool;   // HDI def M 102.4: Safety limit switch top chamber lift
      XT_ROT_CAM_TRG : Bool;   // HDI def M 102.5: limit switch xtal rotation camera trigger
      MP_ENB_K8 : Bool;   // HDI def M 102.6: Mobile panel agree button +K8
      MP_ENB_K9 : Bool;   // HDI def M 102.7: Mobile panel agree button +K9
      LS_V3_OP : Bool;   // HDI def M 103.0: valve position V3 open
      LS_V3_CL : Bool;   // HDI def M 103.1: Valve position V3 closed
      FDR_LS_V3_2_OP : Bool;   // HDI def M 103.2: valve position V3_2 open
      FDR_LS_V3_2_CL : Bool;   // HDI def M 103.3: Valve position V3_2 closed
      LSR_SEN_OBJ_DET : Bool;   // HDI def M 103.4: spare digital input
      SPARE_280_5 : Bool;   // HDI def M 103.5: spare digital input
      SPARE_280_6 : Bool;   // HDI def M 103.6: spare digital input
      SPARE_280_7 : Bool;   // HDI def M 103.7: spare digital input
      LS_V11_OP : Bool;   // HDI def M 89.3: V 11 open (isolation valve feeder)
      LS_V11_CL : Bool;   // HDI def M 89.4: V 11 closed (isolation valve feeder)
      FDR_HOP_CON : Bool;   // HDI def M 89.5: hopper connected to feeder
   END_VAR
BEGIN
END_DATA_BLOCK

DATA_BLOCK "SDO"   // DB132
{ S7_Optimized_Access := 'FALSE' }
VERSION : 0.0
// --------------------------------------------------------------------------------
// program:             SDO
// description :        automatically generated SDO
// name:                hp
// date        :        03.02.2021
// 
// revision:
// name:
// date:
//                     (c)CGS
// --------------------------------------------------------------------------------
   VAR
      HOR_OPP_K2 : Bool;   // HDO def M 136.0: Horn +K2
      LMP_RD_K2 : Bool;   // HDO def M 136.1: Lamp red +K2
      LMP_YE_K2 : Bool;   // HDO def M 136.2: Lamp yellow +K2
      LMP_GN_K2 : Bool;   // HDO def M 136.3: Lamp green +K2
      LMP_BU_K2 : Bool;   // HDO def M 136.4: Lamp blue +K2
      HOR_MAG_ACTIVE : Bool;   // HDO def M 136.5: Horn magnet active( Lift)
      LMP_MAG_ACTIVE : Bool;   // HDO def M 136.6: Lamp magnet active( Lift+ Field on)
      SPARE_16_7 : Bool;   // HDO def M 136.7: spare digital output
      P1_ON : Bool;   // HDO def M 137.0: Vacuum pump 1 on (furnace chamber)
      P3_ON : Bool;   // HDO def M 137.1: Vacuum pump 3 on (gate chamber)
      P2_ON : Bool;   // HDO def M 137.2: Vacuum pump 2 on (roots furnace chamber)
      P1_SEAL_GAS : Bool;   // HDO def M 137.3: Vacuum pump 1 seal gas on
      P3_SEAL_GAS : Bool;   // HDO def M 137.4: Vacuum pump 3 seal gas on
      HTR_PWR_ON : Bool;   // HDO def M 137.4: Heater power supply on
      V10 : Bool;   // HDO def M 137.6: Vacuum pump 1 secuvac valve V10 on
      MON_TMP_P2_RES : Bool;   // HDO def M 137.7: temperature monitoring pump 2 reset
      SPARE_18_0 : Bool;   // HDO def M 138.0: spare digital output
      SPARE_18_1 : Bool;   // HDO def M 138.1: spare digital output
      SPARE_18_2 : Bool;   // HDO def M 138.2: spare digital output
      SPARE_18_3 : Bool;   // HDO def M 138.3: spare digital output
      SPARE_18_4 : Bool;   // HDO def M 138.4: spare digital output
      SPARE_18_5 : Bool;   // HDO def M 138.5: spare digital output
      SPARE_18_6 : Bool;   // HDO def M 138.6: spare digital output
      SPARE_18_7 : Bool;   // HDO def M 138.7: spare digital output
      V1_OP : Bool;   // HDO def M 142.0: V1 open
      V1_CL : Bool;   // HDO def M 142.1: V1 close
      SPARE_32_2 : Bool;   // HDO def M 142.2: spare digital output
      SPARE_32_3 : Bool;   // HDO def M 142.3: spare digital output
      SPARE_32_4 : Bool;   // HDO def M 142.4: spare digital output
      CR_ROT_ENB : Bool;   // HDO def M 142.5: controller enable crucible rotation
      CR_LFT_ENB : Bool;   // HDO def M 142.6: controller enable crucible lift
      FU_FCB_HDL_ON : Bool;   // HDO def M 142.7: Frequency converter FCB handling on
      TEC_FLG_LFT_ENB : Bool;   // HDO def M 143.0: controller enable techn chamber lift
      FCH_LFT_ENB : Bool;   // HDO def M 143.1: controller enable lower chamber parts lift
      MAG_LFT_UP : Bool;   // HDO def M 143.2: Magnet lift drive upwards
      MAG_LFT_DN : Bool;   // HDO def M 143.3: Magnet lift drive downwards
      BRK_MAG_LFT : Bool;   // HDO def M 143.4: Brake magnet lift
      SPARE_33_5 : Bool;   // HDO def M 143.5: spare digital output
      SPARE_33_6 : Bool;   // HDO def M 143.6: spare digital output
      SPARE_33_7 : Bool;   // HDO def M 143.7: spare digital output
      V1_1_OP : Bool;   // HDO def M 144.0: V1.1 open
      V1_1_CL : Bool;   // HDO def M 144.1: V1.1 close
      SPARE_34_2 : Bool;   // HDO def M 144.2: spare digital output
      SPARE_34_3 : Bool;   // HDO def M 144.3: spare digital output
      SPARE_34_4 : Bool;   // HDO def M 144.4: spare digital output
      SPARE_34_5 : Bool;   // HDO def M 144.5: spare digital output
      SPARE_34_6 : Bool;   // HDO def M 144.6: spare digital output
      SPARE_34_7 : Bool;   // HDO def M 144.7: spare digital output
      ACC_SC_HTR_STR : Bool;   // HDO def M 146.0: ACC Heizung START
      ACC_SC_HTR_RST : Bool;   // HDO def M 146.1: ACC Heizung RESET
      ACC_SC_WTR_STR : Bool;   // HDO def M 146.2: ACC K黨lwasser START
      ACC_SC_WTR_RST : Bool;   // HDO def M 146.3: ACC K黨lwasser RESET
      ACC_ALM_LT_1 : Bool;   // HDO def M 146.4: ACC Blitzlicht Kasten
      ACC_ALM_SND_1 : Bool;   // HDO def M 146.5: ACC Sirene Kasten
      ACC_ALM_LT_2 : Bool;   // HDO def M 146.6: ACC Blitzlicht Bedienpult
      ACC_ALM_SND_2 : Bool;   // HDO def M 146.7: ACC Sirene Bedienpult
      FCH_HOOK_HOME : Bool;   // HDO def M 150.0: Valve block lower furnace chamber hook unlocking
      FCH_HOOK_WORK : Bool;   // HDO def M 150.1: Valve block lower furnace chamber hook locking
      UP_FCH_SW_BRK : Bool;   // HDO def M 150.2: Valve block upper chamber swivel release brake
      LO_FCH_SW_BRK : Bool;   // HDO def M 150.3: Valve block lower chamber swivel release brake
      TEC_FLG_SW_BRK : Bool;   // HDO def M 150.4: Valve block tech. flange swivel release brake
      V25 : Bool;   // HDO def M 150.5: Valve block argon inlet pressure storage tank, V25 open
      V2_1 : Bool;   // HDO def M 150.6: Valve block vacuum valve, V2.1 open
      V21 : Bool;   // HDO def M 150.7: Valve block air valve vacuum pipe, V21+V21.1 open
      V19 : Bool;   // HDO def M 151.0: Valve block extraktion valve filter, V19 open
      V20 : Bool;   // HDO def M 151.1: Valve block air valve filter, V20 open
      V22 : Bool;   // HDO def M 151.2: Valve block argon valve filter, V22 open
      V9_2 : Bool;   // HDO def M 151.3: Valve block ventiliation valve vaccum line gate, V9_2
      V22_1 : Bool;   // HDO def M 151.4: Valve block argon valve bypass filter, V22.1 open
      V3_4 : Bool;   // HDO def M 151.5: Valve block vacuum valve, V3.4 open
      V3_3 : Bool;   // HDO def M 151.6: Valve block vacuum valve, V3.3 open
      V2_11 : Bool;   // HDO def M 151.7: Valve block vacuum valve, V2.11 open
      P2_FU_ON : Bool;   // HDO def M 152.0: Frequency converter P2 start
      P2_FU_RES : Bool;   // HDO def M 152.1: Frequency converter P2 fault reset
      SPARE_144_2 : Bool;   // HDO def M 152.2: spare digital output
      SPARE_144_3 : Bool;   // HDO def M 152.3: spare digital output
      SPARE_144_4 : Bool;   // HDO def M 152.4: spare digital output
      SPARE_144_5 : Bool;   // HDO def M 152.5: spare digital output
      SPARE_144_6 : Bool;   // HDO def M 152.6: spare digital output
      SPARE_144_7 : Bool;   // HDO def M 152.7: spare digital output
      V4 : Bool;   // HDO def M 150.0: Valve block V4 valve argon gas inlet (gate chamber)
      V5 : Bool;   // HDO def M 150.1: Valve block V5 valve argon gas inlet controlled (gch)
      V6 : Bool;   // HDO def M 150.2: Valve block V6 valve argon gas inlet controlled (Fch)
      V3 : Bool;   // HDO def M 150.3: Valve block V3 vacuum valve (gate chamber)
      V3_2 : Bool;   // HDO def M 150.4: Valve block V3.2 vacuum valve feeder
      V24 : Bool;   // HDO def M 150.5: Valve block V24 valve argon gas inlet feeder
      XT_DRP_OUT_PRT_CL : Bool;   // HDO def M 150.6: Valve block close crystal drop out protection
      XT_DRP_OUT_PRT_OP : Bool;   // HDO def M 150.7: Valve block open crystal drop out protection
      TCH_SW_LOCK : Bool;   // HDO def M 151.0: Valve block top chamber swivel lock close
      TCH_SW_UNLOCK : Bool;   // HDO def M 151.1: Valve block top chamber swivel lock open
      GCH_SW_LOCK : Bool;   // HDO def M 151.2: Valve block gate chamber swivel lock close
      GCH_SW_UNLOCK : Bool;   // HDO def M 151.3: Valve block gate chamber swivel lock open
      XT_HDL_SW_LOCK : Bool;   // HDO def M 151.4: Valve block xtal handling swivel lock close (145?
      XT_HDL_SW_UNLOCK : Bool;   // HDO def M 151.5: Valve block xtal handling swivel lock open (145?
      FDR_V11_OP : Bool;   // HDO def M 151.6: Valve block open V11 (isolation valve feeder)
      FDR_V11_CL : Bool;   // HDO def M 151.7: Valve block close V11 (isolation valve feeder)
      FDR_V11_CVR_OP : Bool;   // HDO def M 152.0: Valve block open cover V11 (isolation valve feeder)
      FDR_V11_CVR_CL : Bool;   // HDO def M 152.1: Valve block close cover V11 (isolation valve feeder)
      SPARE_226_2 : Bool;   // HDO def M 152.2: Valve block spare output
      SPARE_226_3 : Bool;   // HDO def M 152.3: Valve block spare output
      SPARE_226_4 : Bool;   // HDO def M 152.4: Valve block spare output
      SPARE_226_5 : Bool;   // HDO def M 152.5: Valve block spare output
      SPARE_226_6 : Bool;   // HDO def M 152.6: Valve block spare output
      SPARE_226_7 : Bool;   // HDO def M 152.7: Valve block spare output
      HOR_OPP_K8 : Bool;   // HDO def M 160.0: Horn +K8
      LMP_RD_K8 : Bool;   // HDO def M 160.1: Lamp red +K8
      LMP_YE_K8 : Bool;   // HDO def M 160.2: Lamp yellow +K8
      LMP_GN_K8 : Bool;   // HDO def M 160.3: Lamp green +K8
      LMP_BU_K8 : Bool;   // HDO def M 160.4: Lamp blue +K8
      XT_ROT_ENB : Bool;   // HDO def M 160.5: controller enable crystal rotation
      XT_LFT_ENB : Bool;   // HDO def M 160.6: controller enable crystal lift
      XT_HDL_LFT_ENB : Bool;   // HDO def M 160.7: controller enable crystal handling lift
      XT_HDL_SW_ENB : Bool;   // HDO def M 161.0: controller enable crystal handling swivel
      FU_GCB_HDL_ON : Bool;   // HDO def M 161.1: Frequency converter GCB handling on
      LSR_SEN_PWR_ON : Bool;   // HDO def M 161.2: supply voltage for laser sensor on
      SPARE_273_3 : Bool;   // HDO def M 161.3: spare digital output
      SPARE_273_4 : Bool;   // HDO def M 161.4: spare digital output
      SPARE_273_5 : Bool;   // HDO def M 161.5: spare digital output
      XT_HDL_SLID_FW : Bool;   // HDO def M 161.6: Motor crystal handling slider forwards
      XT_HDL_SLID_BW : Bool;   // HDO def M 161.7: Motor crystal handling slider backwards
      XT_CLP_TILT_BW : Bool;   // HDO def M 163.0: Motor crystal clamp tilt backwards
      XT_CLP_TILT_FW : Bool;   // HDO def M 163.1: Motor crystal clamp tilt forwards (75?
      XT_CLP_TILT_BRK : Bool;   // HDO def M 163.2: Motor crystal clamp tilt brake
      XT_CLP_ABV_OP : Bool;   // HDO def M 163.3: Motor crystal clamp above open
      XT_CLP_ABV_CL : Bool;   // HDO def M 163.4: Motor crystal clamp above close
      XT_CLP_ABV_BRK : Bool;   // HDO def M 163.5: Brake crystal clamp above
      XT_CLP_ABV_RST : Bool;   // HDO def M 163.6: Reset controller crystal clamp above
      GCH_LFT_ENB : Bool;   // HDO def M 163.7: controller enable gate chamber lift
      XT_CLP_BLW_OP : Bool;   // HDO def M 164.0: Motor crystal clamp below open
      XT_CLP_BLW_CL : Bool;   // HDO def M 164.1: Motor crystal clamp below close
      XT_CLP_BLW_BRK : Bool;   // HDO def M 164.2: Brake crystal clamp below
      XT_CLP_BLW_RST : Bool;   // HDO def M 164.3: Reset controller crystal clamp below
      MCC_TEST_XT : Bool;   // HDO def M 164.4: seed contact detection test output ( xt isolated)
      MCC_ENB_XT : Bool;   // HDO def M 164.5: seed contact detection enable output (xt isolated)
      TCH_LFT_ENB : Bool;   // HDO def M 164.6: controller enable top chamber lift
      TCH_TILT_ENB : Bool;   // HDO def M 164.7: controller enable top chamber tilt
      GTE_V_LFT_ENB : Bool;   // HDO def M 165.0: controller enable gate valve lift
      GTE_V_SW_ENB : Bool;   // HDO def M 165.1: controller enable gate valve swivel
      BEL_LFT_ENB : Bool;   // HDO def M 165.2: controller enable gate bellow lift
      HOR_OPP_K9 : Bool;   // HDO def M 165.3: Horn +K9
      LMP_RD_K9 : Bool;   // HDO def M 165.4: Lamp red +K9
      LMP_YE_K9 : Bool;   // HDO def M 165.5: Lamp yellow +K9
      LMP_GN_K9 : Bool;   // HDO def M 165.6: Lamp green +K9
      LMP_BU_K9 : Bool;   // HDO def M 165.7: Lamp blue +K9
   END_VAR
BEGIN
END_DATA_BLOCK

DATA_BLOCK "PAI"   // DB133
{ S7_Optimized_Access := 'FALSE' }
VERSION : 0.0
// --------------------------------------------------------------------------------
// program:             PAI
// description :        automatically generated PAI
// name:                hp
// date        :        03.02.2021
// 
// revision:
// name:
// date:
//                     (c)CGS
// --------------------------------------------------------------------------------
   VAR
      TRV_ACT_POS : Real;   // HAI def MW 192: actual throttle valve position
      TRV_ACT_POS_1 : Real;   // HAI def MW 194: actual throttle valve 1.1 position
      TRV_PRS_FIL_1 : Real;   // HAI def MW 204: actual pressure value main filter
      TRV_PRS_FIL_2 : Real;   // HAI def MW 206: actual pressure value bypass filter
      PYR_ACT_HTR_1_TMP : Real;   // HAI def MW 250: actual temperature main heater
      ACT_PRS_AR_VSL : Real;   // HAI def MW 252: actual pressure argon storage tank
      SPARE_484 : Real;   // HAI def MW 254: spare analog output (4..20 mA)
      SPARE_486 : Real;   // HAI def MW 256: spare analog output (4..20 mA)
      PYR_ACT_MELT_TMP : Real;   // HAI def MW 280: actual temperature melt
      SPARE_1538 : Real;   // HAI def MW 282: spare analog output (4..20 mA)
      SPARE_1540 : Real;   // HAI def MW 284: spare analog output (4..20 mA)
      SPARE_1542 : Real;   // HAI def MW 286: spare analog output (4..20 mA)
      GCH_PCR_ACT_PRS : Real;   // HAI def MW 242: actual vacuum gauge gate chamber 5xe-4...1500 mbar
      FCH_PCR_ACT_PRS : Real;   // HAI def MW 200: actual vacuum gauge furnace chamber 5xe-4...1500 mbar
      FCH_BAR_ACT_PRS_100 : Real;   // HAI def MW 198: actual vacuum gauge furnace chamber 100 mbar
      ACC_WTR_TMP : Real;   // HAI def MW 258: ACC water temp.
      ACC_WTR_PRS_IN : Real;   // HAI def MW 260: ACC water pressure
      ACC_WTR_FLW_OUT : Real;   // HAI def MW 262: ACC waterflow output
      ACC_WTR_FLW_IN : Real;   // HAI def MW 264: ACC waterflow input
      ACC_WTR_SPL_PRS : Real;   // HAI def MW 266: ACC water supply inlet pressure
      ACC_SPARE_810 : Real;   // HAI def MW 268: ACC spare
      SPARE : Real;   // HAI def MW 270: spare
   END_VAR
BEGIN
END_DATA_BLOCK

DATA_BLOCK "PAO"   // DB134
{ S7_Optimized_Access := 'FALSE' }
VERSION : 0.0
// --------------------------------------------------------------------------------
// program:             PAO
// description :        automatically generated PAO
// name:                hp
// date        :        03.02.2021
// 
// revision:
// name:
// date:
//                     (c)CGS
// --------------------------------------------------------------------------------
   VAR
      TRV_SET_POS : Real;   // HAO def MW 300: setpoint throttle valve 1 position
      TRV_SET_POS_1 : Real;   // HAO def MW 302: setpoint throttle valve 1.1 position
      SPARE : Real;   // HAO def MW 304: spare
   END_VAR
BEGIN
END_DATA_BLOCK

DATA_BLOCK "SAI"   // DB135
{ S7_Optimized_Access := 'FALSE' }
VERSION : 0.0
// --------------------------------------------------------------------------------
// program:             SAI
// description :        automatically generated SAI
// name:                hp
// date        :        03.02.2021
// 
// revision:
// name:
// date:
//                     (c)CGS
// --------------------------------------------------------------------------------
   VAR
      TRV_ACT_POS : Real;   // HAI def MW 192: actual throttle valve position
      TRV_ACT_POS_1 : Real;   // HAI def MW 194: actual throttle valve 1.1 position
      TRV_PRS_FIL_1 : Real;   // HAI def MW 204: actual pressure value main filter
      TRV_PRS_FIL_2 : Real;   // HAI def MW 206: actual pressure value bypass filter
      PYR_ACT_HTR_1_TMP : Real;   // HAI def MW 250: actual temperature main heater
      ACT_PRS_AR_VSL : Real;   // HAI def MW 252: actual pressure argon storage tank
      SPARE_484 : Real;   // HAI def MW 254: spare analog output (4..20 mA)
      SPARE_486 : Real;   // HAI def MW 256: spare analog output (4..20 mA)
      PYR_ACT_MELT_TMP : Real;   // HAI def MW 280: actual temperature melt
      SPARE_1538 : Real;   // HAI def MW 282: spare analog output (4..20 mA)
      SPARE_1540 : Real;   // HAI def MW 284: spare analog output (4..20 mA)
      SPARE_1542 : Real;   // HAI def MW 286: spare analog output (4..20 mA)
      GCH_PCR_ACT_PRS : Real;   // HAI def MW 242: actual vacuum gauge gate chamber 5xe-4...1500 mbar
      FCH_PCR_ACT_PRS : Real;   // HAI def MW 200: actual vacuum gauge furnace chamber 5xe-4...1500 mbar
      FCH_BAR_ACT_PRS_100 : Real;   // HAI def MW 198: actual vacuum gauge furnace chamber 100 mbar
      ACC_WTR_TMP : Real;   // HAI def MW 258: ACC water temp.
      ACC_WTR_PRS_IN : Real;   // HAI def MW 260: ACC water pressure
      ACC_WTR_FLW_OUT : Real;   // HAI def MW 262: ACC waterflow output
      ACC_WTR_FLW_IN : Real;   // HAI def MW 264: ACC waterflow input
      ACC_WTR_SPL_PRS : Real;   // HAI def MW 266: ACC water supply inlet pressure
      ACC_SPARE_810 : Real;   // HAI def MW 268: ACC spare
      SPARE : Real;   // HAI def MW 270: spare
   END_VAR
BEGIN
END_DATA_BLOCK

DATA_BLOCK "SAO"   // DB136
{ S7_Optimized_Access := 'FALSE' }
VERSION : 0.0
// --------------------------------------------------------------------------------
// program:             SAO
// description :        automatically generated SAO
// name:                hp
// date        :        03.02.2021
// 
// revision:
// name:
// date:
//                     (c)CGS
// --------------------------------------------------------------------------------
   VAR
      TRV_SET_POS : Real;   // HAO def MW 300: setpoint throttle valve 1 position
      TRV_SET_POS_1 : Real;   // HAO def MW 302: setpoint throttle valve 1.1 position
      SPARE : Real;   // HAO def MW 304: spare
   END_VAR
BEGIN
END_DATA_BLOCK

DATA_BLOCK "DV"   // DB137
{ S7_Optimized_Access := 'FALSE' }
VERSION : 0.0
// --------------------------------------------------------------------------------
//     program     :    DV
//     description :    define all DV values       
//     name        :    K. Kalkowski
//     date        :    26.10.99
// 
//     revision    :    CGS  1218
//     name        :    John Wang
//     date        :    08.11.2018
//                     
//     --------------------------------------------------------------------------------
   VAR
      HND_LFT_UP : Bool;   // byte 0
      HND_LFT_DN : Bool;
      HND_LFT_FAST : Bool;
      HND_LFT_OFF : Bool;
      HND_LS_LFT_UP : Bool;
      HND_LS_LFT_DN : Bool;
      HND_LFT_FST_UP_ENB : Bool;
      HND_LFT_FST_DN_ENB : Bool;
      HND_LS_LFT_UP_STOP : Bool;   // byte 1
      HND_LS_LFT_DN_STOP : Bool;
      HND_LT_LFT_UP : Bool;
      HND_LT_LFT_DN : Bool;
      HND_LT_LFT_FAST : Bool;
      HND_LT_LFT_OFF : Bool;
      HND_LT_LFT_FLT : Bool;
      HND_LFT_STOP_IMM : Bool;
      HND_V9_1_OP_REQ : Bool;   // byte 2
      HND_V9_2_OP_REQ : Bool;
      HTR_ITL_OK : Bool;
      HTR_1_PWR_ENB : Bool;
      CR_ROT_FAST : Bool;
      CR_ROT_OFFS_ON : Bool;
      CR_ROT_CTL_OFFS_RP : Bool;
      CR_ROT_OFFS_RP_START : Bool;
      CAM_MELT_COMPLETE : Bool;   // byte 3
      CAM_DIP_COMPLETE : Bool;
      DI_MCC_CONTACT : Bool;
      MLT_LVL_FND : Bool;
      SET_XT_LFT_REF_POS : Bool;
      SET_CR_LFT_REF_POS : Bool;
      SET_HDL_LFT_REF_POS : Bool;
      DRV_SERVICE : Bool;
      CR_LS_LFT_UP : Bool;   // byte 4
      CR_LS_LFT_DN : Bool;
      CR_LFT_FAST_UP_ENB : Bool;
      CR_LFT_FAST_DN_ENB : Bool;
      XT_LS_LFT_UP : Bool;
      XT_LS_LFT_DN : Bool;
      XT_LFT_FAST_UP_ENB : Bool;
      XT_LFT_FAST_DN_ENB : Bool;
      HND_SWL_IN : Bool;   // byte 5
      HND_SWL_OUT : Bool;
      HND_SWL_FAST : Bool;
      HND_SWL_OFF : Bool;
      HND_LT_SWL_IN : Bool;
      HND_LT_SWL_OUT : Bool;
      HND_LT_SWL_FAST : Bool;
      HND_LT_SWL_OFF : Bool;
      HND_LT_SWL_FLT : Bool;   // byte 6
      HND_GCH_SWL_ENB : Bool;
      HND_V9_CLOSE_REQ : Bool;
      HND_SWL_IN_FINAL : Bool;
      HND_TCH_SWL_ENB : Bool;
      HND_WEIGHT_LIM : Bool;
      HND_FCH_SWL_ENB : Bool;
      V9_2_DLY_OP : Bool;
      MAG_LFT_UP : Bool;   // byte 7
      MAG_LFT_DN : Bool;
      MAG_LFT_FAST : Bool;
      MAG_LFT_OFF : Bool;
      SPARE_7_4 : Bool;
      NE_RESTART : Bool;
      SI_FIL_FSH_SEQ_ON : Bool;
      APS_FIL_DELAYED : Bool;
      APS_FCH_DELAYED : Bool;   // byte 8
      APS_GCH_DELAYED : Bool;
      V5_CLOSE_REQ : Bool;
      V6_CLOSE_REQ : Bool;
      APS_FDR_DELAYED : Bool;
      FDR_AUTO_PMP_DN_ENB : Bool;
      FDR_PMP_DN_REQ : Bool;
      MAIN_SWITCH_ON : Bool;
      CAM_PRD_CHG_OK : Bool;   // byte 9
      CAM_MLT_CHK : Bool;
      CAM_PRD_CHG_OK_DLY : Bool;
      CAM_ISP_ON_OK : Bool;
      CAM_ISP_OFF_OK : Bool;
      CAM_ISP_ON : Bool;
      CAM_INIT : Bool;
      SPARE_9_7 : Bool;
      PWR_FAIL_HTR_OFF : Bool;   // byte 10
      PWR_FAIL_MAG_OFF : Bool;
      PWR_FAIL_XT_ROT_OFF : Bool;
      PWR_FAIL_P1_ON : Bool;
      PWR_FAIL_P2_ON : Bool;
      PWR_FAIL_P3_ON : Bool;
      MAIN_LINE_FAULT : Bool;
      PWR_FAIL_HTR_1_ON : Bool;
      PWR_FAIL_HTR_2_ON : Bool;   // byte 11
      ALARM_ACKN : Bool;
      ALARM_ACKN_OLD : Bool;
      PWR_FAIL_MAG_ON : Bool;
      MAG_1_ON : Bool;
      MAG_2_ON : Bool;
      START_SH_FLAG : Bool;   // flag is set with start of shoulder and reset with growth control on
      TRANS_SH_BY_FLAG : Bool;   // flag is set in transistion TO body period
      THR_CALC_ACTIVE : Bool;   // byte 12
      THR_CALC_DISABLED : Bool;   // flag threshold calculation disabled
      EMG_DVC_OFF : Bool;   // flag to switch off drives and heater when emergency mode active
      EMG_DRV_ENB : Bool;   // flag to enable switches on op panel for xt and cr lift
      EMG_STOP : Bool;
      HOR_OPP : Bool;
      LMP_OR : Bool;
      XT_WGT_CELL_TAR_REQ : Bool;
      PRS_CTRL_STD_ALG : Bool;   // byte 13
      DIA_CTRL_STD_ALG : Bool;
      HTR_1_CTRL_STD_ALG : Bool;
      SPD_CTRL_STD_ALG : Bool;
      CRUC_ROT_CTRL_STD_ALG : Bool;
      MLT_TMP_CTRL_STD_ALG : Bool;
      GRW_RTE_CTRL_STD_ALG : Bool;
      V_OP_DLY_P1 : Bool;
      V_OP_DLY_P2 : Bool;   // byte 14
      V_OP_DLY_P3 : Bool;
      MAIN_LINE_460V_FLT : Bool;
      EXT_DVT_TRG_PRV : Bool;
      SIHI_VAC_OP_ACTIVE : Bool;
      PMP_TO_FIN_PRS : Bool;
      SIHI_RUNNING : Bool;
      SIHI_CTRL_RDY : Bool;
      SIHI_PMP_RDY : Bool;   // byte 15
      HTR_1_PWR_SPL_IN_RMT : Bool;
      HTR_1_PWR_SPL_RUN : Bool;
      RST_EFF_XT_SPD : Bool;
      RST_MAN_OP_TIME_CNT : Bool;
      NEW_SI_CRG_WGT_CALC : Bool;
      SI_FIL_FSH_REQ : Bool;
      FIL_FSH_REQ_AFTER_SD : Bool;
      MOB_FDR_CALL : Bool;
      MOB_FDR_P3_ON_REQ : Bool;
      MOB_FDR_V3_2_OPN_REQ : Bool;
      MOB_FDR_V24_OPN_REQ : Bool;
      MVE_FDR_TUBE_DN : Bool;
      MVE_FDR_TUBE_UP : Bool;
      CB_FLT_AC230V_FDR : Bool;
      CB_FLT_DC24V_FDR : Bool;
      FDR_CH_HOME_POS : Bool;
      FDR_CH_FDG_POS : Bool;
      FDR_TUBE_HOME_POS : Bool;
      FDR_TUBE_FCH_POS : Bool;
      FDR_TUBE_FDG_POS : Bool;
      FDR_IN_POS : Bool;
      FDG_MVE_IN_SEQ_DONE : Bool;
      FDG_MVE_OUT_SEQ_DONE : Bool;
      MOB_FDR_V11_OPN_REQ : Bool;
      MOB_FDR_V11_CLD_REQ : Bool;
      MOB_FDR_V11_INST : Bool;
      MOB_FDR_CON : Bool;
      MOB_FDR_PB_TRM : Bool;
      FDR_CH_SW_R : Bool;
      FDR_CH_SW_L : Bool;
      FDR_VIB_ENB : Bool;
      XT_MEN_CNTR : Bool;
      AUTO_OP_CALL : Bool;
      ACC_INST : Bool;
      ACC_OVP_TEST_ON : Bool;
      ACC_ENB_VAC : Bool;
      MAN_ACKN_XT_RMV : Bool;
      ACC_ENB_GAS_V : Bool;
      FIL_VNT_REQ : Bool;
      DST_MLT_FNL_OK : Bool;
      NEW_MSR_TEL_RECV : Bool;
      ARB_XT_DN_BY_CAM : Bool;
      CRUC_ROT_SMI : Bool;
      HTR_1_SMI : Bool;
      XT_LFT_SMI : Bool;
      SPARE_20_6 : Bool;
      SPARE_20_7 : Bool;
      SPARE_21_0 : Bool;
      SPARE_21_1 : Bool;
      MOB_FDR_KL2552_INIT : Bool;
      FIL_FSH_AUTO_START : Bool;
      MOB_FDR_UDCK_ON : Bool;
      MOB_FDR_HOP_EMP : Bool;
      CALC_STD_DEV_FILL_LVL : Bool;
      SET_IMG_IVG_TRG : Bool;
      SERVICE : Bool;
      V7_OP : Bool;
      V7_CL : Bool;
      LS_V7_UP_DLY : Bool;
      LS_V7_DN_DLY : Bool;
      LS_V7_SW_IN_DLY : Bool;
      LS_V7_SW_OUT_DLY : Bool;
      XT_HDL_SW_SET_REF_POS : Bool;
      FCH_SET_REF_POS : Bool;
      TEC_FLG_SET_REF_POS : Bool;
      LO_FCH_SW_SET_REF_POS : Bool;
      UP_FCH_SW_SET_REF_POS : Bool;
      TEC_FLG_SW_SET_REF_POS : Bool;
      LO_FCH_SW_HOME_POS : Bool;
      UP_FCH_SW_HOME_POS : Bool;
      TEC_FLG_SW_HOME_POS : Bool;
      HOOK_POS_0 : Bool;
      HOOK_POS_90 : Bool;
      LS_XT_HDL_LFT_DN_POS : Bool;
      LS_XT_HDL_LFT_UP_POS : Bool;
      LS_XT_HDL_LFT_UP_MAX_POS : Bool;
      LS_XT_HDL_LFT_TRP_POS : Bool;
      LS_XT_ACP_LFT_MID_POS : Bool;
      LS_XT_ACP_LFT_LWR_POS : Bool;
      LS_XT_ACP_LFT_UPR_POS : Bool;
      LS_XT_HDL_SW_IN_CRU_POS : Bool;
      LS_XT_HDL_SW_IN_XT_POS : Bool;
      LS_XT_HDL_SW_IN_TRP_POS : Bool;
      LS_XT_HDL_SW_OUT_MAX_POS : Bool;
      XT_HDL_SEQ_MOD : Bool;
      LS_XT_HDL_SW_IN_POS : Bool;
      LS_XT_HDL_SW_OUT_POS : Bool;
      MP_SERVICE : Bool;
      APS_BY_FIL_DELAYED : Bool;
      V1_HAND_MODE : Bool;
      V1_1_HAND_MODE : Bool;
      V2_1_CL : Bool;
      V2_11_OP : Bool;
      V3_3_OP : Bool;
      V3_4_OP : Bool;
      V22_1_OP : Bool;
      FIL_CLN_REQ_IN_PRC : Bool;
      S_CAM_RAD_RT_ACTV : Bool;
      CTL_MLT_DRIFT_ON : Bool;
      P3_ON : Bool;
      V22_OP : Bool;
      MAN_XT_LFT_UP : Bool;
      MAN_CR_LFT_UP : Bool;
      V25_OP : Bool;
      P1_GAS_BAL_ENB : Bool;
   END_VAR
BEGIN
END_DATA_BLOCK

DATA_BLOCK "AV"   // DB138
{ S7_Optimized_Access := 'FALSE' }
VERSION : 0.0
// --------------------------------------------------------------------------------
//     program     :    AV
//     description :    define all AV values       
//     name        :    G. Eibelsh鋟ser
//     date        :    26.10.2007
// 
//     revision    :  
//     name        :   
//     date        :    
// 
//                     (c)PVA TePla AG       
//     --------------------------------------------------------------------------------
   VAR
      LRT_EKZ : Real;
      ACT_PRS_FCH : Real;   // actual pressure furnace
      ACT_XT_POS : Real;
      ACT_CR_POS : Real;
      ACT_CR_REF_POS : Real;
      SET_XT_SPD : Real;
      SET_CR_SPD : Real;
      ACT_XT_SPD : Real;
      ACT_CR_SPD : Real;
      SET_XT_POS : Real;
      SET_CR_POS : Real;
      SET_GAS_1_FLW : Real;
      SET_GAS_2_FLW : Real;
      SET_PRS_FCH : Real;
      ACT_PRS_GCH : Real;   // actual pressure gate
      ACT_PRS_FDR : Real;   // actual pressure feeder
      ACT_XT_LEN : Real;
      ACT_XT_LEN_PRC : Real;
      ACT_XT_DIA : Real;
      INP_XT_DIA : Real;
      OUTP_XT_DIA_FIL : Real;
      SET_XT_DIA : Real;
      SET_XT_ROT : Real;
      SET_CR_ROT : Real;
      ACT_XT_ROT : Real;
      ACT_CR_ROT : Real;
      SET_CTL_VALVE_POS : Real;
      ACT_HTR_1_TMP : Real;
      ACT_HTR_2_TMP : Real;
      AVG_HTR_1_TMP : Real;
      AVG_HTR_2_TMP : Real;
      SET_HTR_1_PWR : Real;
      SET_HTR_2_PWR : Real;
      SET_HTR_1_TMP_INC : Real;
      SET_HTR_2_PWR_INC : Real;
      SET_HND_LFT_SPD : Real;   // setpoint handling lift speed
      SET_HND_SWL_SPD : Real;   // setpoint handling swivel speed
      SET_MAG_LFT_SPD : Real;   // setpoint magnet lift speed
      SET_MAG_1_CUR : Real;
      SET_MAG_2_CUR : Real;
      SET_MAG_AV_CUR : Real;
      SET_MAG_RATIO_CUR : Real;
      SET_XT_LEN_BDY2 : Real;
      SET_CR_POS_BDY2 : Real;
      CRUC_RATIO : Real;
      XT_LEN_BY2_RP : Real;
      ACT_HTR_1_RES : Real;   // power supply resistance values
      ACT_HTR_1_RES_CNG : Real;
      ACT_HTR_2_RES : Real;
      ACT_HTR_2_RES_CNG : Real;
      ACT_HTR_3_RES : Real;
      ACT_HTR_3_RES_CNG : Real;
      ACT_MAG_1_RES : Real;
      ACT_MAG_1_RES_CNG : Real;
      ACT_MAG_2_RES : Real;
      ACT_MAG_2_RES_CNG : Real;
      PWR_FAIL_HTR_1_PWR : Real;   // save last power value after power fail
      PWR_FAIL_HTR_2_PWR : Real;
      PWR_FAIL_MAG_1_CUR : Real;
      PWR_FAIL_MAG_2_CUR : Real;
      CR_ROT_OFFS_TIME : Real;   // crucible rot offset on/off time
      ACT_CR_ROT_SET : Real;   // actual crucible rotation setpoint
      CALC_THR : Real;   // calculated threshold value
      SET_MLT_LVL_LSR : Real;
      DIFF_PRS_FDR_FNC : Real;   // difference prs furnace - prs feeder
      ACT_LRT_FDR : Real;   // leak rate feeder
      ACT_PRS_DROP_FDR : Real;   // pressure drop feeder at final V11 test
      ACT_HTR_1_PWR : Real;
      ACT_HTR_1_CUR : Real;
      ACT_HTR_1_VLT : Real;
      ACT_DVT_PRD_NO : Real;
      INP_BGT_AREA : Real;
      INP_BLOBS : Real;
      ACT_XT_WGT_CALC : Real;
      ACT_XT_WGT : Real;
      XT_TAR_WGT : Real;
      ACT_XT_WGT_TAR : Real;
      AVG_XT_WGT_TAR : Real;
      ACT_HTR_2_PWR : Real;
      ACT_HTR_2_CUR : Real;
      ACT_HTR_2_VLT : Real;
      ACT_TOT_XT_LGH : Real;
      ACT_XT_WGT_RTE : Real;
      ACT_XT_DIA_CALC : Real;
      ACT_XT_POS_INC : Real;
      ACT_XT_DIA_CALC_ALT : Real;
      ACT_WTR_TMP_VPTS : Real;
      ACT_WTR_FLW_VPTS : Real;
      ACT_GEAR_OIL_TMP_P1 : Real;
      ACT_COOLANT_TMP_P1 : Real;
      ACT_MAX_CUR_P1 : Real;
      ACT_MAX_CUR_P2 : Real;
      ACT_PRD_2_CTR_X : Real;
      ACT_PRD_2_CTR_Y : Real;
      AVG_PRD_2_CTR_X : Real;
      AVG_PRD_2_CTR_Y : Real;
      ACT_MLT_LVL : Real;
      ACT_MLT_VIB_DIST : Real;
      MOB_FDR_LKR : Real;
      MOB_FDR_ACT_TUBE_TMP : Real;
      MOB_FDR_ACT_TUBE_POS : Real;
      MOB_FDR_ACT_CRG_LVL : Real;
      SET_MOB_FDR_VIB_FRQ : Real;
      SET_FDG_RTE : Real;
      ACT_STB_NE_LEN : Real;
      ACT_STB_NE_LEN_PRC : Real;
      SH_TRS_DIA : Real;
      TOT_GAS_CSP : Real;
      TOT_PWR_CSP : Real;
      ACT_DIA_PTS_INCL : Real;
      SET_DIP_TMP : Real;
      XT_POS_AT_START_BY : Real;
      MLT_LVL_SFT_OFFS_SPD : Real;
      XT_HDL_SW_ENC_POS : Real;
      FCH_ENC_POS : Real;
      TEC_FLG_ENC_POS : Real;
      LO_FCH_SW_ENC_POS : Real;
      UP_FCH_SW_ENC_POS : Real;
      TEC_FLG_SW_ENC_POS : Real;
      XT_HDL_CLP_WGT : Real;
      XT_HDL_CLP_TAR_WGT : Real;
      XT_HDL_LFT_ACT_POS : Real;
      ACT_CRUC_FILL_LVL : Real;
      XT_HDL_SW_ACT_POS : Real;
      INP_CAL_XT_DIA : Real;
      S_CAM_DELTA_R : Real;
      S_CAM_DELTA_H : Real;
      S_CAM_1_ACT_DIA_CF : Real;
      S_CAM_1_AVG_DIA_CF : Real;
      S_CAM_2_ACT_DIA_CF : Real;
      S_CAM_2_AVG_DIA_CF : Real;
      S_CAM_1_ACT_RAD_PT : Real;
      S_CAM_1_AVG_RAD_PT : Real;
      S_CAM_2_ACT_RAD_PT : Real;
      S_CAM_2_AVG_RAD_PT : Real;
      S_CAM_1_ACT_CF_CTR_X : Real;
      S_CAM_1_AVG_CF_CTR_X : Real;
      S_CAM_1_ACT_CF_CTR_Y : Real;
      S_CAM_2_ACT_CF_CTR_X : Real;
      S_CAM_2_AVG_CF_CTR_X : Real;
      S_CAM_2_ACT_CF_CTR_Y : Real;
      S_CAM_ACT_XT_DIA : Real;
      S_CAM_AVG_XT_DIA : Real;
      S_CAM_ACT_MLT_LVL_CHG : Real;
      S_CAM_AVG_MLT_LVL_CHG : Real;
      AVG_XT_DIA : Real;
   END_VAR
BEGIN
END_DATA_BLOCK

DATA_BLOCK "DC"   // DB139
{ S7_Optimized_Access := 'FALSE' }
VERSION : 0.0
// --------------------------------------------------------------------------------
//     program     :    DC
//     description :    define all DC values       
//     name        :    G. Eibelsh鋟ser
//     date        :    26.10.2007
// 
//     revision    :
//     name        :
//     date        :    
//                     (c)PVA TePla AG       
//     --------------------------------------------------------------------------------
   VAR
      MOD_AUT_ENB : Bool;   // word 0
      MOD_ID : Bool;
      MOD_CH : Bool;
      MOD_PD : Bool;
      MOD_ME : Bool;
      MOD_DI : Bool;
      MOD_NE : Bool;
      MOD_SH : Bool;
      MOD_BY : Bool;
      MOD_EC : Bool;
      MOD_RE : Bool;
      MOD_SD : Bool;
      CTL_MLT_1_TMP_ON : Bool;
      CTL_MLT_2_TMP_ON : Bool;
      CTL_DIA_ON : Bool;
      CTL_GRW_RTE_ON : Bool;
      CTL_PULL_RTE_ON : Bool;   // word 1
      CTL_CRUC_ROT_ON : Bool;
      CTL_MLT_LVL_ON : Bool;
      CTL_SI_FDR_ON : Bool;
      CTL_DOP_FDR_ON : Bool;
      XT_LFT_UP : Bool;
      XT_LFT_DN : Bool;
      XT_LFT_FST : Bool;
      XT_ROT_CW : Bool;
      XT_ROT_CCW : Bool;
      CR_LFT_UP : Bool;
      CR_LFT_DN : Bool;
      CR_LFT_FST : Bool;
      CR_ROT_CW : Bool;
      CR_ROT_CCW : Bool;
      HTR_1_ON : Bool;
      CTL_HTR_1_TMP_ON : Bool;   // word 2
      HTR_2_ON : Bool;
      CTL_HTR_2_TMP_ON : Bool;
      HTR_3_ON : Bool;
      MAG_ON : Bool;
      SI_FDR_ON : Bool;
      DOP_FDR_ON : Bool;
      RST_DOP_CNT : Bool;
      CTL_PRS_ON : Bool;
      V1_OP : Bool;
      V2_OP : Bool;
      V3_OP : Bool;
      V4_OP : Bool;
      V5_OP : Bool;
      V6_OP : Bool;
      V8_OP : Bool;
      V11_OP : Bool;   // word 3
      V11_CL : Bool;
      V12_OP : Bool;
      V13_OP : Bool;
      V14_OP : Bool;
      V15_OP : Bool;
      V21_OP : Bool;
      V24_OP : Bool;
      P1_ON : Bool;
      P3_ON : Bool;
      MCC_ON : Bool;
      MCC_TST_ON : Bool;
      LSR_ON : Bool;
      LSR_FIL_HI : Bool;
      CAM_OFF : Bool;
      CAM_MLT : Bool;
      CAM_DIP : Bool;   // word 4
      CAM_DIA : Bool;
      SPARE_8_2 : Bool;
      CAM_SEL_1 : Bool;
      CAM_SEL_2 : Bool;
      CAM_SET_WIN : Bool;
      CAM_SET_THR : Bool;
      V2_1_OP : Bool;
      V2_2_OP : Bool;
      V16_1_OP : Bool;
      V16_2_OP : Bool;
      V1_OPEN_REQ : Bool;
      V1_CLOSE_REQ : Bool;
      SET_HTR_1_TMP_ABS : Bool;
      SET_HTR_2_PWR_ABS : Bool;
      RSTRT_HTR_1_TMP_INC : Bool;
      RSTRT_HTR_2_PWR_INC : Bool;   // word 5
      FDR_FLP_CTL_ON : Bool;
      FDR_FLP_CTL_OFF : Bool;
      FDR_TUBE_DRV_IN : Bool;
      FDR_TUBE_DRV_OUT : Bool;
      V3_2_OP : Bool;
      CAM_ISP_ON : Bool;
      CAM_INIT : Bool;
      P2_ON : Bool;
      V17_OP : Bool;
      V18_OP : Bool;
      V19_OP : Bool;
      V20_OP : Bool;
      V22_OP : Bool;
      V23_OP : Bool;
      V9_1_OP : Bool;
      V25_OP : Bool;   // word 6
      CTL_MLT_DRIFT_ON : Bool;
      V3_0_OP : Bool;
      V3_1_OP : Bool;
      MOB_FDR_MVE_IN_SEQ_ON : Bool;
      MOB_FDR_MVE_OUT_SEQ_ON : Bool;
      MOB_FDR_VIB_ON : Bool;
      XT_HDL_LFT_UP : Bool;
      XT_HDL_LFT_DN : Bool;
      XT_HDL_LFT_FAST : Bool;
      XT_HDL_SW_IN : Bool;
      XT_HDL_SW_OUT : Bool;
      XT_HDL_SW_UNLOCK : Bool;
      XT_HDL_SW_LOCK : Bool;   // word 14
      XT_HDL_SLID_FW : Bool;
      XT_HDL_SLID_BW : Bool;
      XT_CLP_TILT_90 : Bool;
      XT_CLP_TILT_75 : Bool;
      XT_CLP_ABV_OP : Bool;
      XT_CLP_ABV_CL : Bool;
      XT_CLP_BLW_OP : Bool;
      XT_CLP_BLW_CL : Bool;
      OP_XT_DRP_OUT_PRT : Bool;
      CL_XT_DRP_OUT_PRT : Bool;
      V3_4_OP : Bool;
      V1_1_REL : Bool;
      CTL_GAP_ON : Bool;
      CTL_OFFS_SPEED_ON : Bool;
      SPARE_15_7 : Bool;
      RES_ERR_DRV_XT_ROT : Bool;
      ENAB_BM_DRV_XT_ROT : Bool;
      RES_ERR_DRV_CR_ROT : Bool;
      ENAB_BM_DRV_CR_ROT : Bool;
   END_VAR
BEGIN
END_DATA_BLOCK

DATA_BLOCK "AC"   // DB140
{ S7_Optimized_Access := 'FALSE' }
VERSION : 0.0
// --------------------------------------------------------------------------------
//     program     :    AC
//     description :    define all AC values       
//     name        :    G. Eibelsh鋟ser
//     date        :    26.10.2007
// 
//     revision    : 
//     name        :
//     date        :   
//                     (c)PVA TePla AG       
//     --------------------------------------------------------------------------------
   VAR
      SET_XT_SPD : Real;   // word 0
      SET_XT_ROT : Real;
      SET_CR_SPD : Real;
      SET_CR_ROT : Real;
      SET_HTR_1_TMP : Real;
      SET_HTR_2_TMP : Real;
      SET_HTR_1_PWR : Real;
      SET_HTR_2_PWR : Real;
      SET_MLT_1_TMP : Real;   // word 32
      SET_MLT_2_TMP : Real;
      SET_CLF_PRS : Real;
      SET_GAS_1_FLW : Real;
      SET_GAS_2_FLW : Real;
      SET_TRV_POS : Real;
      SET_FDR_SI : Real;
      SET_FDR_DOP : Real;
      SET_CA_THR : Real;   // word 64
      SET_CA_WIN_POS_H : Real;
      SET_CA_WIN_POS_V : Real;
      SET_CA_WIN_SZE_H : Real;
      SET_CA_WIN_SZE_V : Real;
      SET_MLT_LVL_LSR : Real;
      SET_XT_DIA : Real;
      SET_GRW_RTE : Real;
      SET_AVG_SPD : Real;   // word 96
      SET_AVG_CRUC_ROT : Real;
      LVL_AT_STA_BY : Real;
      SET_HTR_1_TMP_INC : Real;
      SET_HTR_2_PWR_INC : Real;
      SET_XT_SPD_DEV_1 : Real;
      SET_XT_SPD_DEV_2 : Real;
      SET_CR_ROT_OFS : Real;
      SET_CR_ROT_ON_TME : Real;   // word 128
      SET_CR_ROT_OFF_TME : Real;
      XT_MENISCUS : Real;
      SET_XT_SPD_INC : Real;
      SET_XT_ROT_INC : Real;
      SET_CR_ROT_INC : Real;
      SET_CR_SPD_COF : Real;
      ACT_NUM_OF_PELLETS : Real;
      MISSING_PELLETS : Real;   // word 160
      SET_CR_SPD_INC : Real;
      SET_HTR_3_PWR : Real;
      SET_MAG_1_CUR : Real;
      SET_MAG_2_CUR : Real;
      SET_MAG_AV_CUR : Real;
      SET_MAG_RATIO_CUR : Real;
      CA_2_PIXEL_FCT : Real;
      CA_2_OFS : Real;
      CR_CHARGE_WGT : Real;
      CR_DIA : Real;
      CR_FILL_LEVEL : Real;
      TMP_COEFF_1 : Real;
      TMP_COEFF_2 : Real;
      PWR_COEFF_1 : Real;
      PWR_COEFF_2 : Real;
      CTL_DIA_GN : Real;
      CTL_DIA_TI : Real;
      CTL_DIA_TD : Real;
      CTL_DIA_T1 : Real;
      CTL_DIA_TF_1 : Real;
      CTL_DIA_TF_2 : Real;
      CTL_GRO_GN : Real;
      CTL_GRO_TI : Real;
      CTL_GRO_TD : Real;
      CTL_GRO_T1 : Real;
      CTL_GRO_TF : Real;
      CTL_AV_SPD_GN : Real;
      CTL_AV_SPD_TI : Real;
      CTL_AV_SPD_TD : Real;
      CTL_AV_SPD_T1 : Real;
      CTL_AV_SPD_TF : Real;
      CTL_AV_CRUC_ROT_GN : Real;
      CTL_AV_CRUC_ROT_TI : Real;
      CTL_AV_CRUC_ROT_TD : Real;
      CTL_AV_CRUC_ROT_T1 : Real;
      CTL_AV_CRUC_ROT_TF : Real;
      CTL_MLT_LVL_GN : Real;
      CTL_MLT_LVL_TI : Real;
      CTL_MLT_LVL_TD : Real;
      CTL_MLT_LVL_T1 : Real;
      CTL_MLT_LVL_TF : Real;
      CTL_MLT_TMP_1_GN : Real;
      CTL_MLT_TMP_1_TI : Real;
      CTL_MLT_TMP_1_TD : Real;
      CTL_MLT_TMP_1_T1 : Real;
      CTL_MLT_TMP_1_TF : Real;
      CTL_PRS_GN : Real;
      CTL_PRS_TI : Real;
      CTL_PRS_TD : Real;
      CTL_PRS_T1 : Real;
      CTL_PRS_TF : Real;
      CTL_HTR_1_TMP_GN : Real;
      CTL_HTR_1_TMP_TI : Real;
      CTL_HTR_1_TMP_TD : Real;
      CTL_HTR_1_TMP_T1 : Real;
      CTL_HTR_1_TMP_TF : Real;
      CTL_HTR_1_AVG_TMP_TF : Real;
      CTL_HTR_2_TMP_GN : Real;
      CTL_HTR_2_TMP_TI : Real;
      CTL_HTR_2_TMP_TD : Real;
      CTL_HTR_2_TMP_T1 : Real;
      CTL_HTR_2_TMP_TF : Real;
      CTL_HTR_2_AVG_TMP_TF : Real;
      SET_CTL_VALVE_POS : Real;
      SET_CRUC_ROT_DEV_1 : Real;
      SET_CRUC_ROT_DEV_2 : Real;
      SET_CR_ROT_RP_TME_UP : Real;
      SET_CR_ROT_RP_TME_DN : Real;
      SET_MLT_LVL_INC : Real;
      SET_SEN_THR : Real;
      SET_SEN_CTR_X : Real;
      SET_SEN_CTR_Y : Real;
      SET_SEN_OUT_RAD : Real;
      SET_SEN_IN_RAD : Real;
      SET_SEN_SEQ_STR_AGL : Real;
      SET_SEN_SEQ_STP_AGL : Real;
      SET_SEN_WDH : Real;
      SET_SEN_HGT : Real;
      SET_MOB_FDR_VIB_FRQ : Real;
      SET_OP_CALL : Real;
      SET_FDG_RTE : Real;
      CTL_DIA_TMP_GN : Real;
      CTL_DIA_TMP_TI : Real;
      CTL_DIA_TMP_TD : Real;
      CTL_DIA_TMP_T1 : Real;
      SET_CTL_VALVE_POS_V1 : Real;
      SET_CTL_VALVE_POS_V1_1 : Real;
      SET_ROI_CTR_X_SCAM : Real;
      SET_ROI_CTR_Y_SCAM : Real;
      SET_CAM_2_THR : Real;
      CTL_GAP_TI : Real;   // Gap CTL
      CTL_GAP_TD : Real;
      CTL_GAP_T1 : Real;
      CTL_GAP_GN : Real;
      CTL_AV_OFFS_TI : Real;   // VAG Speed Offset Controller xtal lift / cruc lift
      CTL_AV_OFFS_GN : Real;
      CTL_AV_OFFS_T1 : Real;
      CTL_AV_OFFS_TD : Real;
      CTL_OFFS_SPEED_TI : Real;
      CTL_OFFS_SPEED_TD : Real;
      CTL_OFFS_SPEED_T1 : Real;
      CTL_OFFS_SPEED_GN : Real;
   END_VAR
BEGIN
END_DATA_BLOCK

